//     PlcTask Inputs/G_IO.arDI[68]/Ch[15] <-> Module 4 (GL20-1600END)/1600END input-bit maping/Digital input CH2-bit7
//     PlcTask Inputs/G_IO.arDI[68]/Ch[1] <-> Module 4 (GL20-1600END)/1600END input-bit maping/Digital input CH1-bit1
//     PlcTask Inputs/G_IO.arDI[68]/Ch[2] <-> Module 4 (GL20-1600END)/1600END input-bit maping/Digital input CH1-bit2
//     PlcTask Inputs/G_IO.arDI[68]/Ch[3] <-> Module 4 (GL20-1600END)/1600END input-bit maping/Digital input CH1-bit3
//     PlcTask Inputs/G_IO.arDI[68]/Ch[4] <-> Module 4 (GL20-1600END)/1600END input-bit maping/Digital input CH1-bit4
//     PlcTask Inputs/G_IO.arDI[68]/Ch[5] <-> Module 4 (GL20-1600END)/1600END input-bit maping/Digital input CH1-bit5
//     PlcTask Inputs/G_IO.arDI[68]/Ch[6] <-> Module 4 (GL20-1600END)/1600END input-bit maping/Digital input CH1-bit6
//     PlcTask Inputs/G_IO.arDI[68]/Ch[7] <-> Module 4 (GL20-1600END)/1600END input-bit maping/Digital input CH1-bit7
//     PlcTask Inputs/G_IO.arDI[68]/Ch[8] <-> Module 4 (GL20-1600END)/1600END input-bit maping/Digital input CH2-bit0
//     PlcTask Inputs/G_IO.arDI[68]/Ch[9] <-> Module 4 (GL20-1600END)/1600END input-bit maping/Digital input CH2-bit1
//     PlcTask Inputs/G_IO.arDI[69]/Ch[0] <-> Module 5 (GL20-1600END)/1600END input-bit maping/Digital input CH1-bit0
//     PlcTask Inputs/G_IO.arDI[69]/Ch[10] <-> Module 5 (GL20-1600END)/1600END input-bit maping/Digital input CH2-bit2
//     PlcTask Inputs/G_IO.arDI[69]/Ch[11] <-> Module 5 (GL20-1600END)/1600END input-bit maping/Digital input CH2-bit3
//     PlcTask Inputs/G_IO.arDI[69]/Ch[12] <-> Module 5 (GL20-1600END)/1600END input-bit maping/Digital input CH2-bit4
//     PlcTask Inputs/G_IO.arDI[69]/Ch[13] <-> Module 5 (GL20-1600END)/1600END input-bit maping/Digital input CH2-bit5
//     PlcTask Inputs/G_IO.arDI[69]/Ch[14] <-> Module 5 (GL20-1600END)/1600END input-bit maping/Digital input CH2-bit6
//     PlcTask Inputs/G_IO.arDI[69]/Ch[15] <-> Module 5 (GL20-1600END)/1600END input-bit maping/Digital input CH2-bit7
//     PlcTask Inputs/G_IO.arDI[69]/Ch[1] <-> Module 5 (GL20-1600END)/1600END input-bit maping/Digital input CH1-bit1
//     PlcTask Inputs/G_IO.arDI[69]/Ch[2] <-> Module 5 (GL20-1600END)/1600END input-bit maping/Digital input CH1-bit2
//     PlcTask Inputs/G_IO.arDI[69]/Ch[3] <-> Module 5 (GL20-1600END)/1600END input-bit maping/Digital input CH1-bit3
//     PlcTask Inputs/G_IO.arDI[69]/Ch[4] <-> Module 5 (GL20-1600END)/1600END input-bit maping/Digital input CH1-bit4
//     PlcTask Inputs/G_IO.arDI[69]/Ch[5] <-> Module 5 (GL20-1600END)/1600END input-bit maping/Digital input CH1-bit5
//     PlcTask Inputs/G_IO.arDI[69]/Ch[6] <-> Module 5 (GL20-1600END)/1600END input-bit maping/Digital input CH1-bit6
//     PlcTask Inputs/G_IO.arDI[69]/Ch[7] <-> Module 5 (GL20-1600END)/1600END input-bit maping/Digital input CH1-bit7
//     PlcTask Inputs/G_IO.arDI[69]/Ch[8] <-> Module 5 (GL20-1600END)/1600END input-bit maping/Digital input CH2-bit0
//     PlcTask Inputs/G_IO.arDI[69]/Ch[9] <-> Module 5 (GL20-1600END)/1600END input-bit maping/Digital input CH2-bit1
//     PlcTask Outputs/G_IO.arDO[62]/Ch[0] <-> Module 6 (GL20-0016ETP)/0016ETP Output-bit maping/Digital output CH1-bit0
//     PlcTask Outputs/G_IO.arDO[62]/Ch[10] <-> Module 6 (GL20-0016ETP)/0016ETP Output-bit maping/Digital output CH2-bit2
//     PlcTask Outputs/G_IO.arDO[62]/Ch[11] <-> Module 6 (GL20-0016ETP)/0016ETP Output-bit maping/Digital output CH2-bit3
//     PlcTask Outputs/G_IO.arDO[62]/Ch[12] <-> Module 6 (GL20-0016ETP)/0016ETP Output-bit maping/Digital output CH2-bit4
//     PlcTask Outputs/G_IO.arDO[62]/Ch[13] <-> Module 6 (GL20-0016ETP)/0016ETP Output-bit maping/Digital output CH2-bit5
//     PlcTask Outputs/G_IO.arDO[62]/Ch[14] <-> Module 6 (GL20-0016ETP)/0016ETP Output-bit maping/Digital output CH2-bit6
//     PlcTask Outputs/G_IO.arDO[62]/Ch[15] <-> Module 6 (GL20-0016ETP)/0016ETP Output-bit maping/Digital output CH2-bit7
//     PlcTask Outputs/G_IO.arDO[62]/Ch[1] <-> Module 6 (GL20-0016ETP)/0016ETP Output-bit maping/Digital output CH1-bit1
//     PlcTask Outputs/G_IO.arDO[62]/Ch[2] <-> Module 6 (GL20-0016ETP)/0016ETP Output-bit maping/Digital output CH1-bit2
//     PlcTask Outputs/G_IO.arDO[62]/Ch[3] <-> Module 6 (GL20-0016ETP)/0016ETP Output-bit maping/Digital output CH1-bit3
//     PlcTask Outputs/G_IO.arDO[62]/Ch[4] <-> Module 6 (GL20-0016ETP)/0016ETP Output-bit maping/Digital output CH1-bit4
//     PlcTask Outputs/G_IO.arDO[62]/Ch[5] <-> Module 6 (GL20-0016ETP)/0016ETP Output-bit maping/Digital output CH1-bit5
//     PlcTask Outputs/G_IO.arDO[62]/Ch[6] <-> Module 6 (GL20-0016ETP)/0016ETP Output-bit maping/Digital output CH1-bit6
//     PlcTask Outputs/G_IO.arDO[62]/Ch[7] <-> Module 6 (GL20-0016ETP)/0016ETP Output-bit maping/Digital output CH1-bit7
//     PlcTask Outputs/G_IO.arDO[62]/Ch[8] <-> Module 6 (GL20-0016ETP)/0016ETP Output-bit maping/Digital output CH2-bit0
//     PlcTask Outputs/G_IO.arDO[62]/Ch[9] <-> Module 6 (GL20-0016ETP)/0016ETP Output-bit maping/Digital output CH2-bit1
//     PlcTask Outputs/G_IO.arDO[63]/Ch[0] <-> Module 7 (GL20-0016ETP)/0016ETP Output-bit maping/Digital output CH1-bit0
//     PlcTask Outputs/G_IO.arDO[63]/Ch[10] <-> Module 7 (GL20-0016ETP)/0016ETP Output-bit maping/Digital output CH2-bit2
//     PlcTask Outputs/G_IO.arDO[63]/Ch[11] <-> Module 7 (GL20-0016ETP)/0016ETP Output-bit maping/Digital output CH2-bit3
//     PlcTask Outputs/G_IO.arDO[63]/Ch[12] <-> Module 7 (GL20-0016ETP)/0016ETP Output-bit maping/Digital output CH2-bit4
//     PlcTask Outputs/G_IO.arDO[63]/Ch[13] <-> Module 7 (GL20-0016ETP)/0016ETP Output-bit maping/Digital output CH2-bit5
//     PlcTask Outputs/G_IO.arDO[63]/Ch[14] <-> Module 7 (GL20-0016ETP)/0016ETP Output-bit maping/Digital output CH2-bit6
//     PlcTask Outputs/G_IO.arDO[63]/Ch[15] <-> Module 7 (GL20-0016ETP)/0016ETP Output-bit maping/Digital output CH2-bit7
//     PlcTask Outputs/G_IO.arDO[63]/Ch[1] <-> Module 7 (GL20-0016ETP)/0016ETP Output-bit maping/Digital output CH1-bit1
//     PlcTask Outputs/G_IO.arDO[63]/Ch[2] <-> Module 7 (GL20-0016ETP)/0016ETP Output-bit maping/Digital output CH1-bit2
//     PlcTask Outputs/G_IO.arDO[63]/Ch[3] <-> Module 7 (GL20-0016ETP)/0016ETP Output-bit maping/Digital output CH1-bit3
//     PlcTask Outputs/G_IO.arDO[63]/Ch[4] <-> Module 7 (GL20-0016ETP)/0016ETP Output-bit maping/Digital output CH1-bit4
//     PlcTask Outputs/G_IO.arDO[63]/Ch[5] <-> Module 7 (GL20-0016ETP)/0016ETP Output-bit maping/Digital output CH1-bit5
//     PlcTask Outputs/G_IO.arDO[63]/Ch[6] <-> Module 7 (GL20-0016ETP)/0016ETP Output-bit maping/Digital output CH1-bit6
//     PlcTask Outputs/G_IO.arDO[63]/Ch[7] <-> Module 7 (GL20-0016ETP)/0016ETP Output-bit maping/Digital output CH1-bit7
//     PlcTask Outputs/G_IO.arDO[63]/Ch[8] <-> Module 7 (GL20-0016ETP)/0016ETP Output-bit maping/Digital output CH2-bit0
//     PlcTask Outputs/G_IO.arDO[63]/Ch[9] <-> Module 7 (GL20-0016ETP)/0016ETP Output-bit maping/Digital output CH2-bit1
//   kittingDeca/kittingDeca Instance <-> pm side/pm6_7_innerConv
//     PlcTask Inputs/GVL.pm[6].inConv.belt[0].fbconverter.running_freq <-> Axis#1 Iutputs/Axis1 Running frequency
//     PlcTask Inputs/GVL.pm[6].inConv.belt[1].fbconverter.running_freq <-> Axis#2 Iutputs/Axis2 Running frequency
//     PlcTask Inputs/GVL.pm[6].inConv.belt[2].fbconverter.running_freq <-> Axis#3 Iutputs/Axis3 Running frequency
//     PlcTask Inputs/GVL.pm[7].inConv.belt[0].fbconverter.running_freq <-> Axis#4 Iutputs/Axis4 Running frequency
//     PlcTask Inputs/GVL.pm[7].inConv.belt[1].fbconverter.running_freq <-> Axis#5 Iutputs/Axis5 Running frequency
//     PlcTask Inputs/GVL.pm[7].inConv.belt[2].fbconverter.running_freq <-> Axis#6 Iutputs/Axis6 Running frequency
//     PlcTask Inputs/GVL.pm[6].inConv.belt[0].fbconverter.status <-> Axis#1 Iutputs/Axis1 AC drive running status word 2
//     PlcTask Inputs/GVL.pm[6].inConv.belt[1].fbconverter.status <-> Axis#2 Iutputs/Axis2 AC drive running status word 2
//     PlcTask Inputs/GVL.pm[6].inConv.belt[2].fbconverter.status <-> Axis#3 Iutputs/Axis3 AC drive running status word 2
//     PlcTask Inputs/GVL.pm[7].inConv.belt[0].fbconverter.status <-> Axis#4 Iutputs/Axis4 AC drive running status word 2
//     PlcTask Inputs/GVL.pm[7].inConv.belt[1].fbconverter.status <-> Axis#5 Iutputs/Axis5 AC drive running status word 2
//     PlcTask Inputs/GVL.pm[7].inConv.belt[2].fbconverter.status <-> Axis#6 Iutputs/Axis6 AC drive running status word 2
//     PlcTask Outputs/GVL.pm[6].inConv.belt[0].fbconverter.cmd <-> Axis#1 Outputs/Axis1 Communication control command
//     PlcTask Outputs/GVL.pm[6].inConv.belt[1].fbconverter.cmd <-> Axis#2 Outputs/Axis2 Communication control command
//     PlcTask Outputs/GVL.pm[6].inConv.belt[2].fbconverter.cmd <-> Axis#3 Outputs/Axis3 Communication control command
//     PlcTask Outputs/GVL.pm[7].inConv.belt[0].fbconverter.cmd <-> Axis#4 Outputs/Axis4 Communication control command
//     PlcTask Outputs/GVL.pm[7].inConv.belt[1].fbconverter.cmd <-> Axis#5 Outputs/Axis5 Communication control command
//     PlcTask Outputs/GVL.pm[7].inConv.belt[2].fbconverter.cmd <-> Axis#6 Outputs/Axis6 Communication control command
//     PlcTask Outputs/GVL.pm[6].inConv.belt[0].fbconverter.freq <-> Axis#1 Outputs/Axis1 Frequency set through communication
//     PlcTask Outputs/GVL.pm[6].inConv.belt[1].fbconverter.freq <-> Axis#2 Outputs/Axis2 Frequency set through communication
//     PlcTask Outputs/GVL.pm[6].inConv.belt[2].fbconverter.freq <-> Axis#3 Outputs/Axis3 Frequency set through communication
//     PlcTask Outputs/GVL.pm[7].inConv.belt[0].fbconverter.freq <-> Axis#4 Outputs/Axis4 Frequency set through communication
//     PlcTask Outputs/GVL.pm[7].inConv.belt[1].fbconverter.freq <-> Axis#5 Outputs/Axis5 Frequency set through communication
//     PlcTask Outputs/GVL.pm[7].inConv.belt[2].fbconverter.freq <-> Axis#6 Outputs/Axis6 Frequency set through communication
//   kittingDeca/kittingDeca Instance <-> pm side/pm6_7_outerConv
//     PlcTask Inputs/GVL.pm[6].outConv.belt[0].fbconverter.running_freq <-> Axis#1 Iutputs/Axis1 Running frequency
//     PlcTask Inputs/GVL.pm[6].outConv.belt[1].fbconverter.running_freq <-> Axis#2 Iutputs/Axis2 Running frequency
//     PlcTask Inputs/GVL.pm[7].outConv.belt[0].fbconverter.running_freq <-> Axis#3 Iutputs/Axis3 Running frequency
//     PlcTask Inputs/GVL.pm[7].outConv.belt[1].fbconverter.running_freq <-> Axis#4 Iutputs/Axis4 Running frequency
//     PlcTask Inputs/GVL.pm[6].outConv.belt[0].fbconverter.status <-> Axis#1 Iutputs/Axis1 AC drive running status word 2
//     PlcTask Inputs/GVL.pm[6].outConv.belt[1].fbconverter.status <-> Axis#2 Iutputs/Axis2 AC drive running status word 2
//     PlcTask Inputs/GVL.pm[7].outConv.belt[0].fbconverter.status <-> Axis#3 Iutputs/Axis3 AC drive running status word 2
//     PlcTask Inputs/GVL.pm[7].outConv.belt[1].fbconverter.status <-> Axis#4 Iutputs/Axis4 AC drive running status word 2
//     PlcTask Outputs/GVL.pm[6].outConv.belt[0].fbconverter.cmd <-> Axis#1 Outputs/Axis1 Communication control command
//     PlcTask Outputs/GVL.pm[6].outConv.belt[1].fbconverter.cmd <-> Axis#2 Outputs/Axis2 Communication control command
//     PlcTask Outputs/GVL.pm[7].outConv.belt[0].fbconverter.cmd <-> Axis#3 Outputs/Axis3 Communication control command
//     PlcTask Outputs/GVL.pm[7].outConv.belt[1].fbconverter.cmd <-> Axis#4 Outputs/Axis4 Communication control command
//     PlcTask Outputs/GVL.pm[6].outConv.belt[0].fbconverter.freq <-> Axis#1 Outputs/Axis1 Frequency set through communication
//     PlcTask Outputs/GVL.pm[6].outConv.belt[1].fbconverter.freq <-> Axis#2 Outputs/Axis2 Frequency set through communication
//     PlcTask Outputs/GVL.pm[7].outConv.belt[0].fbconverter.freq <-> Axis#3 Outputs/Axis3 Frequency set through communication
//     PlcTask Outputs/GVL.pm[7].outConv.belt[1].fbconverter.freq <-> Axis#4 Outputs/Axis4 Frequency set through communication
//   kittingDeca/kittingDeca Instance <-> pm side/pm8_9_dio
//     PlcTask Inputs/G_IO.arDI[70]/Ch[0] <-> Module 1 (GL20-1600END)/1600END input-bit maping/Digital input CH1-bit0
//     PlcTask Inputs/G_IO.arDI[70]/Ch[10] <-> Module 1 (GL20-1600END)/1600END input-bit maping/Digital input CH2-bit2
//     PlcTask Inputs/G_IO.arDI[70]/Ch[11] <-> Module 1 (GL20-1600END)/1600END input-bit maping/Digital input CH2-bit3
//     PlcTask Inputs/G_IO.arDI[70]/Ch[12] <-> Module 1 (GL20-1600END)/1600END input-bit maping/Digital input CH2-bit4
//     PlcTask Inputs/G_IO.arDI[70]/Ch[13] <-> Module 1 (GL20-1600END)/1600END input-bit maping/Digital input CH2-bit5
//     PlcTask Inputs/G_IO.arDI[70]/Ch[14] <-> Module 1 (GL20-1600END)/1600END input-bit maping/Digital input CH2-bit6
//     PlcTask Inputs/G_IO.arDI[70]/Ch[15] <-> Module 1 (GL20-1600END)/1600END input-bit maping/Digital input CH2-bit7
//     PlcTask Inputs/G_IO.arDI[70]/Ch[1] <-> Module 1 (GL20-1600END)/1600END input-bit maping/Digital input CH1-bit1
//     PlcTask Inputs/G_IO.arDI[70]/Ch[2] <-> Module 1 (GL20-1600END)/1600END input-bit maping/Digital input CH1-bit2
//     PlcTask Inputs/G_IO.arDI[70]/Ch[3] <-> Module 1 (GL20-1600END)/1600END input-bit maping/Digital input CH1-bit3
//     PlcTask Inputs/G_IO.arDI[70]/Ch[4] <-> Module 1 (GL20-1600END)/1600END input-bit maping/Digital input CH1-bit4
//     PlcTask Inputs/G_IO.arDI[70]/Ch[5] <-> Module 1 (GL20-1600END)/1600END input-bit maping/Digital input CH1-bit5
//     PlcTask Inputs/G_IO.arDI[70]/Ch[6] <-> Module 1 (GL20-1600END)/1600END input-bit maping/Digital input CH1-bit6
//     PlcTask Inputs/G_IO.arDI[70]/Ch[7] <-> Module 1 (GL20-1600END)/1600END input-bit maping/Digital input CH1-bit7
//     PlcTask Inputs/G_IO.arDI[70]/Ch[8] <-> Module 1 (GL20-1600END)/1600END input-bit maping/Digital input CH2-bit0
//     PlcTask Inputs/G_IO.arDI[70]/Ch[9] <-> Module 1 (GL20-1600END)/1600END input-bit maping/Digital input CH2-bit1
//     PlcTask Inputs/G_IO.arDI[71]/Ch[0] <-> Module 2 (GL20-1600END)/1600END input-bit maping/Digital input CH1-bit0
//     PlcTask Inputs/G_IO.arDI[71]/Ch[10] <-> Module 2 (GL20-1600END)/1600END input-bit maping/Digital input CH2-bit2
//     PlcTask Inputs/G_IO.arDI[71]/Ch[11] <-> Module 2 (GL20-1600END)/1600END input-bit maping/Digital input CH2-bit3
//     PlcTask Inputs/G_IO.arDI[71]/Ch[12] <-> Module 2 (GL20-1600END)/1600END input-bit maping/Digital input CH2-bit4
//     PlcTask Inputs/G_IO.arDI[71]/Ch[13] <-> Module 2 (GL20-1600END)/1600END input-bit maping/Digital input CH2-bit5
//     PlcTask Inputs/G_IO.arDI[71]/Ch[14] <-> Module 2 (GL20-1600END)/1600END input-bit maping/Digital input CH2-bit6
//     PlcTask Inputs/G_IO.arDI[71]/Ch[15] <-> Module 2 (GL20-1600END)/1600END input-bit maping/Digital input CH2-bit7
//     PlcTask Inputs/G_IO.arDI[71]/Ch[1] <-> Module 2 (GL20-1600END)/1600END input-bit maping/Digital input CH1-bit1
//     PlcTask Inputs/G_IO.arDI[71]/Ch[2] <-> Module 2 (GL20-1600END)/1600END input-bit maping/Digital input CH1-bit2
//     PlcTask Inputs/G_IO.arDI[71]/Ch[3] <-> Module 2 (GL20-1600END)/1600END input-bit maping/Digital input CH1-bit3
//     PlcTask Inputs/G_IO.arDI[71]/Ch[4] <-> Module 2 (GL20-1600END)/1600END input-bit maping/Digital input CH1-bit4
//     PlcTask Inputs/G_IO.arDI[71]/Ch[5] <-> Module 2 (GL20-1600END)/1600END input-bit maping/Digital input CH1-bit5
//     PlcTask Inputs/G_IO.arDI[71]/Ch[6] <-> Module 2 (GL20-1600END)/1600END input-bit maping/Digital input CH1-bit6
//     PlcTask Inputs/G_IO.arDI[71]/Ch[7] <-> Module 2 (GL20-1600END)/1600END input-bit maping/Digital input CH1-bit7
//     PlcTask Inputs/G_IO.arDI[71]/Ch[8] <-> Module 2 (GL20-1600END)/1600END input-bit maping/Digital input CH2-bit0
//     PlcTask Inputs/G_IO.arDI[71]/Ch[9] <-> Module 2 (GL20-1600END)/1600END input-bit maping/Digital input CH2-bit1
//     PlcTask Inputs/G_IO.arDI[72]/Ch[0] <-> Module 3 (GL20-1600END)/1600END input-bit maping/Digital input CH1-bit0
//     PlcTask Inputs/G_IO.arDI[72]/Ch[10] <-> Module 3 (GL20-1600END)/1600END input-bit maping/Digital input CH2-bit2
//     PlcTask Inputs/G_IO.arDI[72]/Ch[11] <-> Module 3 (GL20-1600END)/1600END input-bit maping/Digital input CH2-bit3
//     PlcTask Inputs/G_IO.arDI[72]/Ch[12] <-> Module 3 (GL20-1600END)/1600END input-bit maping/Digital input CH2-bit4
//     PlcTask Inputs/G_IO.arDI[72]/Ch[13] <-> Module 3 (GL20-1600END)/1600END input-bit maping/Digital input CH2-bit5
//     PlcTask Inputs/G_IO.arDI[72]/Ch[14] <-> Module 3 (GL20-1600END)/1600END input-bit maping/Digital input CH2-bit6
//     PlcTask Inputs/G_IO.arDI[72]/Ch[15] <-> Module 3 (GL20-1600END)/1600END input-bit maping/Digital input CH2-bit7
//     PlcTask Inputs/G_IO.arDI[72]/Ch[1] <-> Module 3 (GL20-1600END)/1600END input-bit maping/Digital input CH1-bit1
//     PlcTask Inputs/G_IO.arDI[72]/Ch[2] <-> Module 3 (GL20-1600END)/1600END input-bit maping/Digital input CH1-bit2
//     PlcTask Inputs/G_IO.arDI[72]/Ch[3] <-> Module 3 (GL20-1600END)/1600END input-bit maping/Digital input CH1-bit3
//     PlcTask Inputs/G_IO.arDI[72]/Ch[4] <-> Module 3 (GL20-1600END)/1600END input-bit maping/Digital input CH1-bit4
//     PlcTask Inputs/G_IO.arDI[72]/Ch[5] <-> Module 3 (GL20-1600END)/1600END input-bit maping/Digital input CH1-bit5
//     PlcTask Inputs/G_IO.arDI[72]/Ch[6] <-> Module 3 (GL20-1600END)/1600END input-bit maping/Digital input CH1-bit6
//     PlcTask Inputs/G_IO.arDI[72]/Ch[7] <-> Module 3 (GL20-1600END)/1600END input-bit maping/Digital input CH1-bit7
//     PlcTask Inputs/G_IO.arDI[72]/Ch[8] <-> Module 3 (GL20-1600END)/1600END input-bit maping/Digital input CH2-bit0
//     PlcTask Inputs/G_IO.arDI[72]/Ch[9] <-> Module 3 (GL20-1600END)/1600END input-bit maping/Digital input CH2-bit1
//     PlcTask Inputs/G_IO.arDI[73]/Ch[0] <-> Module 4 (GL20-1600END)/1600END input-bit maping/Digital input CH1-bit0
//     PlcTask Inputs/G_IO.arDI[73]/Ch[10] <-> Module 4 (GL20-1600END)/1600END input-bit maping/Digital input CH2-bit2
//     PlcTask Inputs/G_IO.arDI[73]/Ch[11] <-> Module 4 (GL20-1600END)/1600END input-bit maping/Digital input CH2-bit3
//     PlcTask Inputs/G_IO.arDI[73]/Ch[12] <-> Module 4 (GL20-1600END)/1600END input-bit maping/Digital input CH2-bit4
//     PlcTask Inputs/G_IO.arDI[73]/Ch[13] <-> Module 4 (GL20-1600END)/1600END input-bit maping/Digital input CH2-bit5
//     PlcTask Inputs/G_IO.arDI[73]/Ch[14] <-> Module 4 (GL20-1600END)/1600END input-bit maping/Digital input CH2-bit6
//     PlcTask Inputs/G_IO.arDI[73]/Ch[15] <-> Module 4 (GL20-1600END)/1600END input-bit maping/Digital input CH2-bit7
//     PlcTask Inputs/G_IO.arDI[73]/Ch[1] <-> Module 4 (GL20-1600END)/1600END input-bit maping/Digital input CH1-bit1
//     PlcTask Inputs/G_IO.arDI[73]/Ch[2] <-> Module 4 (GL20-1600END)/1600END input-bit maping/Digital input CH1-bit2
//     PlcTask Inputs/G_IO.arDI[73]/Ch[3] <-> Module 4 (GL20-1600END)/1600END input-bit maping/Digital input CH1-bit3
//     PlcTask Inputs/G_IO.arDI[73]/Ch[4] <-> Module 4 (GL20-1600END)/1600END input-bit maping/Digital input CH1-bit4
//     PlcTask Inputs/G_IO.arDI[73]/Ch[5] <-> Module 4 (GL20-1600END)/1600END input-bit maping/Digital input CH1-bit5
//     PlcTask Inputs/G_IO.arDI[73]/Ch[6] <-> Module 4 (GL20-1600END)/1600END input-bit maping/Digital input CH1-bit6
//     PlcTask Inputs/G_IO.arDI[73]/Ch[7] <-> Module 4 (GL20-1600END)/1600END input-bit maping/Digital input CH1-bit7
//     PlcTask Inputs/G_IO.arDI[73]/Ch[8] <-> Module 4 (GL20-1600END)/1600END input-bit maping/Digital input CH2-bit0
//     PlcTask Inputs/G_IO.arDI[73]/Ch[9] <-> Module 4 (GL20-1600END)/1600END input-bit maping/Digital input CH2-bit1
//     PlcTask Inputs/G_IO.arDI[74]/Ch[0] <-> Module 5 (GL20-1600END)/1600END input-bit maping/Digital input CH1-bit0
//     PlcTask Inputs/G_IO.arDI[74]/Ch[10] <-> Module 5 (GL20-1600END)/1600END input-bit maping/Digital input CH2-bit2
//     PlcTask Inputs/G_IO.arDI[74]/Ch[11] <-> Module 5 (GL20-1600END)/1600END input-bit maping/Digital input CH2-bit3
//     PlcTask Inputs/G_IO.arDI[74]/Ch[12] <-> Module 5 (GL20-1600END)/1600END input-bit maping/Digital input CH2-bit4
//     PlcTask Inputs/G_IO.arDI[74]/Ch[13] <-> Module 5 (GL20-1600END)/1600END input-bit maping/Digital input CH2-bit5
//     PlcTask Inputs/G_IO.arDI[74]/Ch[14] <-> Module 5 (GL20-1600END)/1600END input-bit maping/Digital input CH2-bit6
//     PlcTask Inputs/G_IO.arDI[74]/Ch[15] <-> Module 5 (GL20-1600END)/1600END input-bit maping/Digital input CH2-bit7
//     PlcTask Inputs/G_IO.arDI[74]/Ch[1] <-> Module 5 (GL20-1600END)/1600END input-bit maping/Digital input CH1-bit1
//     PlcTask Inputs/G_IO.arDI[74]/Ch[2] <-> Module 5 (GL20-1600END)/1600END input-bit maping/Digital input CH1-bit2
//     PlcTask Inputs/G_IO.arDI[74]/Ch[3] <-> Module 5 (GL20-1600END)/1600END input-bit maping/Digital input CH1-bit3
//     PlcTask Inputs/G_IO.arDI[74]/Ch[4] <-> Module 5 (GL20-1600END)/1600END input-bit maping/Digital input CH1-bit4
//     PlcTask Inputs/G_IO.arDI[74]/Ch[5] <-> Module 5 (GL20-1600END)/1600END input-bit maping/Digital input CH1-bit5
//     PlcTask Inputs/G_IO.arDI[74]/Ch[6] <-> Module 5 (GL20-1600END)/1600END input-bit maping/Digital input CH1-bit6
//     PlcTask Inputs/G_IO.arDI[74]/Ch[7] <-> Module 5 (GL20-1600END)/1600END input-bit maping/Digital input CH1-bit7
//     PlcTask Inputs/G_IO.arDI[74]/Ch[8] <-> Module 5 (GL20-1600END)/1600END input-bit maping/Digital input CH2-bit0
//     PlcTask Inputs/G_IO.arDI[74]/Ch[9] <-> Module 5 (GL20-1600END)/1600END input-bit maping/Digital input CH2-bit1
//     PlcTask Outputs/G_IO.arDO[66]/Ch[0] <-> Module 6 (GL20-0016ETP)/0016ETP Output-bit maping/Digital output CH1-bit0
//     PlcTask Outputs/G_IO.arDO[66]/Ch[10] <-> Module 6 (GL20-0016ETP)/0016ETP Output-bit maping/Digital output CH2-bit2
//     PlcTask Outputs/G_IO.arDO[66]/Ch[11] <-> Module 6 (GL20-0016ETP)/0016ETP Output-bit maping/Digital output CH2-bit3
//     PlcTask Outputs/G_IO.arDO[66]/Ch[12] <-> Module 6 (GL20-0016ETP)/0016ETP Output-bit maping/Digital output CH2-bit4
//     PlcTask Outputs/G_IO.arDO[66]/Ch[13] <-> Module 6 (GL20-0016ETP)/0016ETP Output-bit maping/Digital output CH2-bit5
//     PlcTask Outputs/G_IO.arDO[66]/Ch[14] <-> Module 6 (GL20-0016ETP)/0016ETP Output-bit maping/Digital output CH2-bit6
//     PlcTask Outputs/G_IO.arDO[66]/Ch[15] <-> Module 6 (GL20-0016ETP)/0016ETP Output-bit maping/Digital output CH2-bit7
//     PlcTask Outputs/G_IO.arDO[66]/Ch[1] <-> Module 6 (GL20-0016ETP)/0016ETP Output-bit maping/Digital output CH1-bit1
//     PlcTask Outputs/G_IO.arDO[66]/Ch[2] <-> Module 6 (GL20-0016ETP)/0016ETP Output-bit maping/Digital output CH1-bit2
//     PlcTask Outputs/G_IO.arDO[66]/Ch[3] <-> Module 6 (GL20-0016ETP)/0016ETP Output-bit maping/Digital output CH1-bit3
//     PlcTask Outputs/G_IO.arDO[66]/Ch[4] <-> Module 6 (GL20-0016ETP)/0016ETP Output-bit maping/Digital output CH1-bit4
//     PlcTask Outputs/G_IO.arDO[66]/Ch[5] <-> Module 6 (GL20-0016ETP)/0016ETP Output-bit maping/Digital output CH1-bit5
//     PlcTask Outputs/G_IO.arDO[66]/Ch[6] <-> Module 6 (GL20-0016ETP)/0016ETP Output-bit maping/Digital output CH1-bit6
//     PlcTask Outputs/G_IO.arDO[66]/Ch[7] <-> Module 6 (GL20-0016ETP)/0016ETP Output-bit maping/Digital output CH1-bit7
//     PlcTask Outputs/G_IO.arDO[66]/Ch[8] <-> Module 6 (GL20-0016ETP)/0016ETP Output-bit maping/Digital output CH2-bit0
//     PlcTask Outputs/G_IO.arDO[66]/Ch[9] <-> Module 6 (GL20-0016ETP)/0016ETP Output-bit maping/Digital output CH2-bit1
//     PlcTask Outputs/G_IO.arDO[67]/Ch[0] <-> Module 7 (GL20-0016ETP)/0016ETP Output-bit maping/Digital output CH1-bit0
//     PlcTask Outputs/G_IO.arDO[67]/Ch[10] <-> Module 7 (GL20-0016ETP)/0016ETP Output-bit maping/Digital output CH2-bit2
//     PlcTask Outputs/G_IO.arDO[67]/Ch[11] <-> Module 7 (GL20-0016ETP)/0016ETP Output-bit maping/Digital output CH2-bit3
//     PlcTask Outputs/G_IO.arDO[67]/Ch[12] <-> Module 7 (GL20-0016ETP)/0016ETP Output-bit maping/Digital output CH2-bit4
//     PlcTask Outputs/G_IO.arDO[67]/Ch[13] <-> Module 7 (GL20-0016ETP)/0016ETP Output-bit maping/Digital output CH2-bit5
//     PlcTask Outputs/G_IO.arDO[67]/Ch[14] <-> Module 7 (GL20-0016ETP)/0016ETP Output-bit maping/Digital output CH2-bit6
//     PlcTask Outputs/G_IO.arDO[67]/Ch[15] <-> Module 7 (GL20-0016ETP)/0016ETP Output-bit maping/Digital output CH2-bit7
//     PlcTask Outputs/G_IO.arDO[67]/Ch[1] <-> Module 7 (GL20-0016ETP)/0016ETP Output-bit maping/Digital output CH1-bit1
//     PlcTask Outputs/G_IO.arDO[67]/Ch[2] <-> Module 7 (GL20-0016ETP)/0016ETP Output-bit maping/Digital output CH1-bit2
//     PlcTask Outputs/G_IO.arDO[67]/Ch[3] <-> Module 7 (GL20-0016ETP)/0016ETP Output-bit maping/Digital output CH1-bit3
//     PlcTask Outputs/G_IO.arDO[67]/Ch[4] <-> Module 7 (GL20-0016ETP)/0016ETP Output-bit maping/Digital output CH1-bit4
//     PlcTask Outputs/G_IO.arDO[67]/Ch[5] <-> Module 7 (GL20-0016ETP)/0016ETP Output-bit maping/Digital output CH1-bit5
//     PlcTask Outputs/G_IO.arDO[67]/Ch[6] <-> Module 7 (GL20-0016ETP)/0016ETP Output-bit maping/Digital output CH1-bit6
//     PlcTask Outputs/G_IO.arDO[67]/Ch[7] <-> Module 7 (GL20-0016ETP)/0016ETP Output-bit maping/Digital output CH1-bit7
//     PlcTask Outputs/G_IO.arDO[67]/Ch[8] <-> Module 7 (GL20-0016ETP)/0016ETP Output-bit maping/Digital output CH2-bit0
//     PlcTask Outputs/G_IO.arDO[67]/Ch[9] <-> Module 7 (GL20-0016ETP)/0016ETP Output-bit maping/Digital output CH2-bit1
//   kittingDeca/kittingDeca Instance <-> pm side/pm8_9_innerConv
//     PlcTask Inputs/GVL.pm[8].inConv.belt[0].fbconverter.running_freq <-> Axis#1 Iutputs/Axis1 Running frequency
//     PlcTask Inputs/GVL.pm[8].inConv.belt[1].fbconverter.running_freq <-> Axis#2 Iutputs/Axis2 Running frequency
//     PlcTask Inputs/GVL.pm[8].inConv.belt[2].fbconverter.running_freq <-> Axis#3 Iutputs/Axis3 Running frequency
//     PlcTask Inputs/GVL.pm[9].inConv.belt[0].fbconverter.running_freq <-> Axis#4 Iutputs/Axis4 Running frequency
//     PlcTask Inputs/GVL.pm[9].inConv.belt[1].fbconverter.running_freq <-> Axis#5 Iutputs/Axis5 Running frequency
//     PlcTask Inputs/GVL.pm[9].inConv.belt[2].fbconverter.running_freq <-> Axis#6 Iutputs/Axis6 Running frequency
//     PlcTask Inputs/GVL.pm[8].inConv.belt[0].fbconverter.status <-> Axis#1 Iutputs/Axis1 AC drive running status word 2
//     PlcTask Inputs/GVL.pm[8].inConv.belt[1].fbconverter.status <-> Axis#2 Iutputs/Axis2 AC drive running status word 2
//     PlcTask Inputs/GVL.pm[8].inConv.belt[2].fbconverter.status <-> Axis#3 Iutputs/Axis3 AC drive running status word 2
//     PlcTask Inputs/GVL.pm[9].inConv.belt[0].fbconverter.status <-> Axis#4 Iutputs/Axis4 AC drive running status word 2
//     PlcTask Inputs/GVL.pm[9].inConv.belt[1].fbconverter.status <-> Axis#5 Iutputs/Axis5 AC drive running status word 2
//     PlcTask Inputs/GVL.pm[9].inConv.belt[2].fbconverter.status <-> Axis#6 Iutputs/Axis6 AC drive running status word 2
//     PlcTask Outputs/GVL.pm[8].inConv.belt[0].fbconverter.cmd <-> Axis#1 Outputs/Axis1 Communication control command
//     PlcTask Outputs/GVL.pm[8].inConv.belt[1].fbconverter.cmd <-> Axis#2 Outputs/Axis2 Communication control command
//     PlcTask Outputs/GVL.pm[8].inConv.belt[2].fbconverter.cmd <-> Axis#3 Outputs/Axis3 Communication control command
//     PlcTask Outputs/GVL.pm[9].inConv.belt[0].fbconverter.cmd <-> Axis#4 Outputs/Axis4 Communication control command
//     PlcTask Outputs/GVL.pm[9].inConv.belt[1].fbconverter.cmd <-> Axis#5 Outputs/Axis5 Communication control command
//     PlcTask Outputs/GVL.pm[9].inConv.belt[2].fbconverter.cmd <-> Axis#6 Outputs/Axis6 Communication control command
//     PlcTask Outputs/GVL.pm[8].inConv.belt[0].fbconverter.freq <-> Axis#1 Outputs/Axis1 Frequency set through communication
//     PlcTask Outputs/GVL.pm[8].inConv.belt[1].fbconverter.freq <-> Axis#2 Outputs/Axis2 Frequency set through communication
//     PlcTask Outputs/GVL.pm[8].inConv.belt[2].fbconverter.freq <-> Axis#3 Outputs/Axis3 Frequency set through communication
//     PlcTask Outputs/GVL.pm[9].inConv.belt[0].fbconverter.freq <-> Axis#4 Outputs/Axis4 Frequency set through communication
//     PlcTask Outputs/GVL.pm[9].inConv.belt[1].fbconverter.freq <-> Axis#5 Outputs/Axis5 Frequency set through communication
//     PlcTask Outputs/GVL.pm[9].inConv.belt[2].fbconverter.freq <-> Axis#6 Outputs/Axis6 Frequency set through communication
//   kittingDeca/kittingDeca Instance <-> pm side/pm8_9_outerConv
//     PlcTask Inputs/GVL.pm[8].outConv.belt[0].fbconverter.running_freq <-> Axis#1 Iutputs/Axis1 Running frequency
//     PlcTask Inputs/GVL.pm[8].outConv.belt[1].fbconverter.running_freq <-> Axis#2 Iutputs/Axis2 Running frequency
//     PlcTask Inputs/GVL.pm[9].outConv.belt[0].fbconverter.running_freq <-> Axis#3 Iutputs/Axis3 Running frequency
//     PlcTask Inputs/GVL.pm[9].outConv.belt[1].fbconverter.running_freq <-> Axis#4 Iutputs/Axis4 Running frequency
//     PlcTask Inputs/GVL.pm[8].outConv.belt[0].fbconverter.status <-> Axis#1 Iutputs/Axis1 AC drive running status word 2
//     PlcTask Inputs/GVL.pm[8].outConv.belt[1].fbconverter.status <-> Axis#2 Iutputs/Axis2 AC drive running status word 2
//     PlcTask Inputs/GVL.pm[9].outConv.belt[0].fbconverter.status <-> Axis#3 Iutputs/Axis3 AC drive running status word 2
//     PlcTask Inputs/GVL.pm[9].outConv.belt[1].fbconverter.status <-> Axis#4 Iutputs/Axis4 AC drive running status word 2
//     PlcTask Outputs/GVL.pm[8].outConv.belt[0].fbconverter.cmd <-> Axis#1 Outputs/Axis1 Communication control command
//     PlcTask Outputs/GVL.pm[8].outConv.belt[1].fbconverter.cmd <-> Axis#2 Outputs/Axis2 Communication control command
//     PlcTask Outputs/GVL.pm[9].outConv.belt[0].fbconverter.cmd <-> Axis#3 Outputs/Axis3 Communication control command
//     PlcTask Outputs/GVL.pm[9].outConv.belt[1].fbconverter.cmd <-> Axis#4 Outputs/Axis4 Communication control command
//     PlcTask Outputs/GVL.pm[8].outConv.belt[0].fbconverter.freq <-> Axis#1 Outputs/Axis1 Frequency set through communication
//     PlcTask Outputs/GVL.pm[8].outConv.belt[1].fbconverter.freq <-> Axis#2 Outputs/Axis2 Frequency set through communication
//     PlcTask Outputs/GVL.pm[9].outConv.belt[0].fbconverter.freq <-> Axis#3 Outputs/Axis3 Frequency set through communication
//     PlcTask Outputs/GVL.pm[9].outConv.belt[1].fbconverter.freq <-> Axis#4 Outputs/Axis4 Frequency set through communication
//   kittingDeca/kittingDeca Instance <-> rem_wf/mcp_dio
//     PlcTask Inputs/G_IO.arDI[95]/Ch[0] <-> Module 1 (GL20-1600END)/1600END input-bit maping/Digital input CH1-bit0
//     PlcTask Inputs/G_IO.arDI[95]/Ch[10] <-> Module 1 (GL20-1600END)/1600END input-bit maping/Digital input CH2-bit2
//     PlcTask Inputs/G_IO.arDI[95]/Ch[11] <-> Module 1 (GL20-1600END)/1600END input-bit maping/Digital input CH2-bit3
//     PlcTask Inputs/G_IO.arDI[95]/Ch[12] <-> Module 1 (GL20-1600END)/1600END input-bit maping/Digital input CH2-bit4
//     PlcTask Inputs/G_IO.arDI[95]/Ch[13] <-> Module 1 (GL20-1600END)/1600END input-bit maping/Digital input CH2-bit5
//     PlcTask Inputs/G_IO.arDI[95]/Ch[14] <-> Module 1 (GL20-1600END)/1600END input-bit maping/Digital input CH2-bit6
//     PlcTask Inputs/G_IO.arDI[95]/Ch[15] <-> Module 1 (GL20-1600END)/1600END input-bit maping/Digital input CH2-bit7
//     PlcTask Inputs/G_IO.arDI[95]/Ch[1] <-> Module 1 (GL20-1600END)/1600END input-bit maping/Digital input CH1-bit1
//     PlcTask Inputs/G_IO.arDI[95]/Ch[2] <-> Module 1 (GL20-1600END)/1600END input-bit maping/Digital input CH1-bit2
//     PlcTask Inputs/G_IO.arDI[95]/Ch[3] <-> Module 1 (GL20-1600END)/1600END input-bit maping/Digital input CH1-bit3
//     PlcTask Inputs/G_IO.arDI[95]/Ch[4] <-> Module 1 (GL20-1600END)/1600END input-bit maping/Digital input CH1-bit4
//     PlcTask Inputs/G_IO.arDI[95]/Ch[5] <-> Module 1 (GL20-1600END)/1600END input-bit maping/Digital input CH1-bit5
//     PlcTask Inputs/G_IO.arDI[95]/Ch[6] <-> Module 1 (GL20-1600END)/1600END input-bit maping/Digital input CH1-bit6
//     PlcTask Inputs/G_IO.arDI[95]/Ch[7] <-> Module 1 (GL20-1600END)/1600END input-bit maping/Digital input CH1-bit7
//     PlcTask Inputs/G_IO.arDI[95]/Ch[8] <-> Module 1 (GL20-1600END)/1600END input-bit maping/Digital input CH2-bit0
//     PlcTask Inputs/G_IO.arDI[95]/Ch[9] <-> Module 1 (GL20-1600END)/1600END input-bit maping/Digital input CH2-bit1
//     PlcTask Outputs/G_IO.arDO[95]/Ch[0] <-> Module 2 (GL20-0016ETP)/0016ETP Output-bit maping/Digital output CH1-bit0
//     PlcTask Outputs/G_IO.arDO[95]/Ch[10] <-> Module 2 (GL20-0016ETP)/0016ETP Output-bit maping/Digital output CH2-bit2
//     PlcTask Outputs/G_IO.arDO[95]/Ch[11] <-> Module 2 (GL20-0016ETP)/0016ETP Output-bit maping/Digital output CH2-bit3
//     PlcTask Outputs/G_IO.arDO[95]/Ch[12] <-> Module 2 (GL20-0016ETP)/0016ETP Output-bit maping/Digital output CH2-bit4
//     PlcTask Outputs/G_IO.arDO[95]/Ch[13] <-> Module 2 (GL20-0016ETP)/0016ETP Output-bit maping/Digital output CH2-bit5
//     PlcTask Outputs/G_IO.arDO[95]/Ch[14] <-> Module 2 (GL20-0016ETP)/0016ETP Output-bit maping/Digital output CH2-bit6
//     PlcTask Outputs/G_IO.arDO[95]/Ch[15] <-> Module 2 (GL20-0016ETP)/0016ETP Output-bit maping/Digital output CH2-bit7
//     PlcTask Outputs/G_IO.arDO[95]/Ch[1] <-> Module 2 (GL20-0016ETP)/0016ETP Output-bit maping/Digital output CH1-bit1
//     PlcTask Outputs/G_IO.arDO[95]/Ch[2] <-> Module 2 (GL20-0016ETP)/0016ETP Output-bit maping/Digital output CH1-bit2
//     PlcTask Outputs/G_IO.arDO[95]/Ch[3] <-> Module 2 (GL20-0016ETP)/0016ETP Output-bit maping/Digital output CH1-bit3
//     PlcTask Outputs/G_IO.arDO[95]/Ch[4] <-> Module 2 (GL20-0016ETP)/0016ETP Output-bit maping/Digital output CH1-bit4
//     PlcTask Outputs/G_IO.arDO[95]/Ch[5] <-> Module 2 (GL20-0016ETP)/0016ETP Output-bit maping/Digital output CH1-bit5
//     PlcTask Outputs/G_IO.arDO[95]/Ch[6] <-> Module 2 (GL20-0016ETP)/0016ETP Output-bit maping/Digital output CH1-bit6
//     PlcTask Outputs/G_IO.arDO[95]/Ch[7] <-> Module 2 (GL20-0016ETP)/0016ETP Output-bit maping/Digital output CH1-bit7
//     PlcTask Outputs/G_IO.arDO[95]/Ch[8] <-> Module 2 (GL20-0016ETP)/0016ETP Output-bit maping/Digital output CH2-bit0
//     PlcTask Outputs/G_IO.arDO[95]/Ch[9] <-> Module 2 (GL20-0016ETP)/0016ETP Output-bit maping/Digital output CH2-bit1
//   kittingDeca/kittingDeca Instance <-> rem_wf/rem0_dio
//     PlcTask Inputs/G_IO.arDI[0]/Ch[0] <-> DI0/1600END input-bit maping/Digital input CH1-bit0
//     PlcTask Inputs/G_IO.arDI[0]/Ch[10] <-> DI0/1600END input-bit maping/Digital input CH2-bit2
//     PlcTask Inputs/G_IO.arDI[0]/Ch[11] <-> DI0/1600END input-bit maping/Digital input CH2-bit3
//     PlcTask Inputs/G_IO.arDI[0]/Ch[12] <-> DI0/1600END input-bit maping/Digital input CH2-bit4
//     PlcTask Inputs/G_IO.arDI[0]/Ch[13] <-> DI0/1600END input-bit maping/Digital input CH2-bit5
//     PlcTask Inputs/G_IO.arDI[0]/Ch[14] <-> DI0/1600END input-bit maping/Digital input CH2-bit6
//     PlcTask Inputs/G_IO.arDI[0]/Ch[15] <-> DI0/1600END input-bit maping/Digital input CH2-bit7
//     PlcTask Inputs/G_IO.arDI[0]/Ch[1] <-> DI0/1600END input-bit maping/Digital input CH1-bit1
//     PlcTask Inputs/G_IO.arDI[0]/Ch[2] <-> DI0/1600END input-bit maping/Digital input CH1-bit2
//     PlcTask Inputs/G_IO.arDI[0]/Ch[3] <-> DI0/1600END input-bit maping/Digital input CH1-bit3
//     PlcTask Inputs/G_IO.arDI[0]/Ch[4] <-> DI0/1600END input-bit maping/Digital input CH1-bit4
//     PlcTask Inputs/G_IO.arDI[0]/Ch[5] <-> DI0/1600END input-bit maping/Digital input CH1-bit5
//     PlcTask Inputs/G_IO.arDI[0]/Ch[6] <-> DI0/1600END input-bit maping/Digital input CH1-bit6
//     PlcTask Inputs/G_IO.arDI[0]/Ch[7] <-> DI0/1600END input-bit maping/Digital input CH1-bit7
//     PlcTask Inputs/G_IO.arDI[0]/Ch[8] <-> DI0/1600END input-bit maping/Digital input CH2-bit0
//     PlcTask Inputs/G_IO.arDI[0]/Ch[9] <-> DI0/1600END input-bit maping/Digital input CH2-bit1
//     PlcTask Inputs/G_IO.arDI[1]/Ch[0] <-> DI1/1600END input-bit maping/Digital input CH1-bit0
//     PlcTask Inputs/G_IO.arDI[1]/Ch[10] <-> DI1/1600END input-bit maping/Digital input CH2-bit2
//     PlcTask Inputs/G_IO.arDI[1]/Ch[11] <-> DI1/1600END input-bit maping/Digital input CH2-bit3
//     PlcTask Inputs/G_IO.arDI[1]/Ch[12] <-> DI1/1600END input-bit maping/Digital input CH2-bit4
//     PlcTask Inputs/G_IO.arDI[1]/Ch[13] <-> DI1/1600END input-bit maping/Digital input CH2-bit5
//     PlcTask Inputs/G_IO.arDI[1]/Ch[14] <-> DI1/1600END input-bit maping/Digital input CH2-bit6
//     PlcTask Inputs/G_IO.arDI[1]/Ch[15] <-> DI1/1600END input-bit maping/Digital input CH2-bit7
//     PlcTask Inputs/G_IO.arDI[1]/Ch[1] <-> DI1/1600END input-bit maping/Digital input CH1-bit1
//     PlcTask Inputs/G_IO.arDI[1]/Ch[2] <-> DI1/1600END input-bit maping/Digital input CH1-bit2
//     PlcTask Inputs/G_IO.arDI[1]/Ch[3] <-> DI1/1600END input-bit maping/Digital input CH1-bit3
//     PlcTask Inputs/G_IO.arDI[1]/Ch[4] <-> DI1/1600END input-bit maping/Digital input CH1-bit4
//     PlcTask Inputs/G_IO.arDI[1]/Ch[5] <-> DI1/1600END input-bit maping/Digital input CH1-bit5
//     PlcTask Inputs/G_IO.arDI[1]/Ch[6] <-> DI1/1600END input-bit maping/Digital input CH1-bit6
//     PlcTask Inputs/G_IO.arDI[1]/Ch[7] <-> DI1/1600END input-bit maping/Digital input CH1-bit7
//     PlcTask Inputs/G_IO.arDI[1]/Ch[8] <-> DI1/1600END input-bit maping/Digital input CH2-bit0
//     PlcTask Inputs/G_IO.arDI[1]/Ch[9] <-> DI1/1600END input-bit maping/Digital input CH2-bit1
//     PlcTask Inputs/G_IO.arDI[2]/Ch[0] <-> DI2/1600END input-bit maping/Digital input CH1-bit0
//     PlcTask Inputs/G_IO.arDI[2]/Ch[10] <-> DI2/1600END input-bit maping/Digital input CH2-bit2
//     PlcTask Inputs/G_IO.arDI[2]/Ch[11] <-> DI2/1600END input-bit maping/Digital input CH2-bit3
//     PlcTask Inputs/G_IO.arDI[2]/Ch[12] <-> DI2/1600END input-bit maping/Digital input CH2-bit4
//     PlcTask Inputs/G_IO.arDI[2]/Ch[13] <-> DI2/1600END input-bit maping/Digital input CH2-bit5
//     PlcTask Inputs/G_IO.arDI[2]/Ch[14] <-> DI2/1600END input-bit maping/Digital input CH2-bit6
//     PlcTask Inputs/G_IO.arDI[2]/Ch[15] <-> DI2/1600END input-bit maping/Digital input CH2-bit7
//     PlcTask Inputs/G_IO.arDI[2]/Ch[1] <-> DI2/1600END input-bit maping/Digital input CH1-bit1
//     PlcTask Inputs/G_IO.arDI[2]/Ch[2] <-> DI2/1600END input-bit maping/Digital input CH1-bit2
//     PlcTask Inputs/G_IO.arDI[2]/Ch[3] <-> DI2/1600END input-bit maping/Digital input CH1-bit3
//     PlcTask Inputs/G_IO.arDI[2]/Ch[4] <-> DI2/1600END input-bit maping/Digital input CH1-bit4
//     PlcTask Inputs/G_IO.arDI[2]/Ch[5] <-> DI2/1600END input-bit maping/Digital input CH1-bit5
//     PlcTask Inputs/G_IO.arDI[2]/Ch[6] <-> DI2/1600END input-bit maping/Digital input CH1-bit6
//     PlcTask Inputs/G_IO.arDI[2]/Ch[7] <-> DI2/1600END input-bit maping/Digital input CH1-bit7
//     PlcTask Inputs/G_IO.arDI[2]/Ch[8] <-> DI2/1600END input-bit maping/Digital input CH2-bit0
//     PlcTask Inputs/G_IO.arDI[2]/Ch[9] <-> DI2/1600END input-bit maping/Digital input CH2-bit1
//     PlcTask Inputs/G_IO.arDI[3]/Ch[0] <-> DI3/1600END input-bit maping/Digital input CH1-bit0
//     PlcTask Inputs/G_IO.arDI[3]/Ch[10] <-> DI3/1600END input-bit maping/Digital input CH2-bit2
//     PlcTask Inputs/G_IO.arDI[3]/Ch[11] <-> DI3/1600END input-bit maping/Digital input CH2-bit3
//     PlcTask Inputs/G_IO.arDI[3]/Ch[12] <-> DI3/1600END input-bit maping/Digital input CH2-bit4
//     PlcTask Inputs/G_IO.arDI[3]/Ch[13] <-> DI3/1600END input-bit maping/Digital input CH2-bit5
//     PlcTask Inputs/G_IO.arDI[3]/Ch[14] <-> DI3/1600END input-bit maping/Digital input CH2-bit6
//     PlcTask Inputs/G_IO.arDI[3]/Ch[15] <-> DI3/1600END input-bit maping/Digital input CH2-bit7
//     PlcTask Inputs/G_IO.arDI[3]/Ch[1] <-> DI3/1600END input-bit maping/Digital input CH1-bit1
//     PlcTask Inputs/G_IO.arDI[3]/Ch[2] <-> DI3/1600END input-bit maping/Digital input CH1-bit2
//     PlcTask Inputs/G_IO.arDI[3]/Ch[3] <-> DI3/1600END input-bit maping/Digital input CH1-bit3
//     PlcTask Inputs/G_IO.arDI[3]/Ch[4] <-> DI3/1600END input-bit maping/Digital input CH1-bit4
//     PlcTask Inputs/G_IO.arDI[3]/Ch[5] <-> DI3/1600END input-bit maping/Digital input CH1-bit5
//     PlcTask Inputs/G_IO.arDI[3]/Ch[6] <-> DI3/1600END input-bit maping/Digital input CH1-bit6
//     PlcTask Inputs/G_IO.arDI[3]/Ch[7] <-> DI3/1600END input-bit maping/Digital input CH1-bit7
//     PlcTask Inputs/G_IO.arDI[3]/Ch[8] <-> DI3/1600END input-bit maping/Digital input CH2-bit0
//     PlcTask Inputs/G_IO.arDI[3]/Ch[9] <-> DI3/1600END input-bit maping/Digital input CH2-bit1
//     PlcTask Outputs/G_IO.arDO[0]/Ch[0] <-> DO0/0016ETP Output-bit maping/Digital output CH1-bit0
//     PlcTask Outputs/G_IO.arDO[0]/Ch[10] <-> DO0/0016ETP Output-bit maping/Digital output CH2-bit2
//     PlcTask Outputs/G_IO.arDO[0]/Ch[11] <-> DO0/0016ETP Output-bit maping/Digital output CH2-bit3
//     PlcTask Outputs/G_IO.arDO[0]/Ch[12] <-> DO0/0016ETP Output-bit maping/Digital output CH2-bit4
//     PlcTask Outputs/G_IO.arDO[0]/Ch[13] <-> DO0/0016ETP Output-bit maping/Digital output CH2-bit5
//     PlcTask Outputs/G_IO.arDO[0]/Ch[14] <-> DO0/0016ETP Output-bit maping/Digital output CH2-bit6
//     PlcTask Outputs/G_IO.arDO[0]/Ch[15] <-> DO0/0016ETP Output-bit maping/Digital output CH2-bit7
//     PlcTask Outputs/G_IO.arDO[0]/Ch[1] <-> DO0/0016ETP Output-bit maping/Digital output CH1-bit1
//     PlcTask Outputs/G_IO.arDO[0]/Ch[2] <-> DO0/0016ETP Output-bit maping/Digital output CH1-bit2
//     PlcTask Outputs/G_IO.arDO[0]/Ch[3] <-> DO0/0016ETP Output-bit maping/Digital output CH1-bit3
//     PlcTask Outputs/G_IO.arDO[0]/Ch[4] <-> DO0/0016ETP Output-bit maping/Digital output CH1-bit4
//     PlcTask Outputs/G_IO.arDO[0]/Ch[5] <-> DO0/0016ETP Output-bit maping/Digital output CH1-bit5
//     PlcTask Outputs/G_IO.arDO[0]/Ch[6] <-> DO0/0016ETP Output-bit maping/Digital output CH1-bit6
//     PlcTask Outputs/G_IO.arDO[0]/Ch[7] <-> DO0/0016ETP Output-bit maping/Digital output CH1-bit7
//     PlcTask Outputs/G_IO.arDO[0]/Ch[8] <-> DO0/0016ETP Output-bit maping/Digital output CH2-bit0
//     PlcTask Outputs/G_IO.arDO[0]/Ch[9] <-> DO0/0016ETP Output-bit maping/Digital output CH2-bit1
//     PlcTask Outputs/G_IO.arDO[1]/Ch[0] <-> DO1/0016ETP Output-bit maping/Digital output CH1-bit0
//     PlcTask Outputs/G_IO.arDO[1]/Ch[10] <-> DO1/0016ETP Output-bit maping/Digital output CH2-bit2
//     PlcTask Outputs/G_IO.arDO[1]/Ch[11] <-> DO1/0016ETP Output-bit maping/Digital output CH2-bit3
//     PlcTask Outputs/G_IO.arDO[1]/Ch[12] <-> DO1/0016ETP Output-bit maping/Digital output CH2-bit4
//     PlcTask Outputs/G_IO.arDO[1]/Ch[13] <-> DO1/0016ETP Output-bit maping/Digital output CH2-bit5
//     PlcTask Outputs/G_IO.arDO[1]/Ch[14] <-> DO1/0016ETP Output-bit maping/Digital output CH2-bit6
//     PlcTask Outputs/G_IO.arDO[1]/Ch[15] <-> DO1/0016ETP Output-bit maping/Digital output CH2-bit7
//     PlcTask Outputs/G_IO.arDO[1]/Ch[1] <-> DO1/0016ETP Output-bit maping/Digital output CH1-bit1
//     PlcTask Outputs/G_IO.arDO[1]/Ch[2] <-> DO1/0016ETP Output-bit maping/Digital output CH1-bit2
//     PlcTask Outputs/G_IO.arDO[1]/Ch[3] <-> DO1/0016ETP Output-bit maping/Digital output CH1-bit3
//     PlcTask Outputs/G_IO.arDO[1]/Ch[4] <-> DO1/0016ETP Output-bit maping/Digital output CH1-bit4
//     PlcTask Outputs/G_IO.arDO[1]/Ch[5] <-> DO1/0016ETP Output-bit maping/Digital output CH1-bit5
//     PlcTask Outputs/G_IO.arDO[1]/Ch[6] <-> DO1/0016ETP Output-bit maping/Digital output CH1-bit6
//     PlcTask Outputs/G_IO.arDO[1]/Ch[7] <-> DO1/0016ETP Output-bit maping/Digital output CH1-bit7
//     PlcTask Outputs/G_IO.arDO[1]/Ch[8] <-> DO1/0016ETP Output-bit maping/Digital output CH2-bit0
//     PlcTask Outputs/G_IO.arDO[1]/Ch[9] <-> DO1/0016ETP Output-bit maping/Digital output CH2-bit1
//   kittingDeca/kittingDeca Instance <-> rem_wf/rem0_valve
//     PlcTask Outputs/G_IO.arDO[2]/Ch[0] <-> Module 1 (C2S-EC-24B)/Outputs/valve[1..4][0]
//     PlcTask Outputs/G_IO.arDO[2]/Ch[10] <-> Module 1 (C2S-EC-24B)/Outputs/valve[5..8][2]
//     PlcTask Outputs/G_IO.arDO[2]/Ch[11] <-> Module 1 (C2S-EC-24B)/Outputs/valve[5..8][3]
//     PlcTask Outputs/G_IO.arDO[2]/Ch[12] <-> Module 1 (C2S-EC-24B)/Outputs/valve[5..8][4]
//     PlcTask Outputs/G_IO.arDO[2]/Ch[13] <-> Module 1 (C2S-EC-24B)/Outputs/valve[5..8][5]
//     PlcTask Outputs/G_IO.arDO[2]/Ch[14] <-> Module 1 (C2S-EC-24B)/Outputs/valve[5..8][6]
//     PlcTask Outputs/G_IO.arDO[2]/Ch[15] <-> Module 1 (C2S-EC-24B)/Outputs/valve[5..8][7]
//     PlcTask Outputs/G_IO.arDO[2]/Ch[1] <-> Module 1 (C2S-EC-24B)/Outputs/valve[1..4][1]
//     PlcTask Outputs/G_IO.arDO[2]/Ch[2] <-> Module 1 (C2S-EC-24B)/Outputs/valve[1..4][2]
//     PlcTask Outputs/G_IO.arDO[2]/Ch[3] <-> Module 1 (C2S-EC-24B)/Outputs/valve[1..4][3]
//     PlcTask Outputs/G_IO.arDO[2]/Ch[4] <-> Module 1 (C2S-EC-24B)/Outputs/valve[1..4][4]
//     PlcTask Outputs/G_IO.arDO[2]/Ch[5] <-> Module 1 (C2S-EC-24B)/Outputs/valve[1..4][5]
//     PlcTask Outputs/G_IO.arDO[2]/Ch[6] <-> Module 1 (C2S-EC-24B)/Outputs/valve[1..4][6]
//     PlcTask Outputs/G_IO.arDO[2]/Ch[7] <-> Module 1 (C2S-EC-24B)/Outputs/valve[1..4][7]
//     PlcTask Outputs/G_IO.arDO[2]/Ch[8] <-> Module 1 (C2S-EC-24B)/Outputs/valve[5..8][0]
//     PlcTask Outputs/G_IO.arDO[2]/Ch[9] <-> Module 1 (C2S-EC-24B)/Outputs/valve[5..8][1]
//     PlcTask Outputs/G_IO.arDO[3]/Ch[0] <-> Module 1 (C2S-EC-24B)/Outputs/valve[9..12][0]
//     PlcTask Outputs/G_IO.arDO[3]/Ch[1] <-> Module 1 (C2S-EC-24B)/Outputs/valve[9..12][1]
//     PlcTask Outputs/G_IO.arDO[3]/Ch[2] <-> Module 1 (C2S-EC-24B)/Outputs/valve[9..12][2]
//     PlcTask Outputs/G_IO.arDO[3]/Ch[3] <-> Module 1 (C2S-EC-24B)/Outputs/valve[9..12][3]
//     PlcTask Outputs/G_IO.arDO[3]/Ch[4] <-> Module 1 (C2S-EC-24B)/Outputs/valve[9..12][4]
//     PlcTask Outputs/G_IO.arDO[3]/Ch[5] <-> Module 1 (C2S-EC-24B)/Outputs/valve[9..12][5]
//     PlcTask Outputs/G_IO.arDO[3]/Ch[6] <-> Module 1 (C2S-EC-24B)/Outputs/valve[9..12][6]
//     PlcTask Outputs/G_IO.arDO[3]/Ch[7] <-> Module 1 (C2S-EC-24B)/Outputs/valve[9..12][7]
//   kittingDeca/kittingDeca Instance <-> rem_wf/rem1_dio
//     PlcTask Inputs/G_IO.arDI[4]/Ch[0] <-> DI4/1600END input-bit maping/Digital input CH1-bit0
//     PlcTask Inputs/G_IO.arDI[4]/Ch[10] <-> DI4/1600END input-bit maping/Digital input CH2-bit2
//     PlcTask Inputs/G_IO.arDI[4]/Ch[11] <-> DI4/1600END input-bit maping/Digital input CH2-bit3
//     PlcTask Inputs/G_IO.arDI[4]/Ch[12] <-> DI4/1600END input-bit maping/Digital input CH2-bit4
//     PlcTask Inputs/G_IO.arDI[4]/Ch[13] <-> DI4/1600END input-bit maping/Digital input CH2-bit5
//     PlcTask Inputs/G_IO.arDI[4]/Ch[14] <-> DI4/1600END input-bit maping/Digital input CH2-bit6
//     PlcTask Inputs/G_IO.arDI[4]/Ch[15] <-> DI4/1600END input-bit maping/Digital input CH2-bit7
//     PlcTask Inputs/G_IO.arDI[4]/Ch[1] <-> DI4/1600END input-bit maping/Digital input CH1-bit1
//     PlcTask Inputs/G_IO.arDI[4]/Ch[2] <-> DI4/1600END input-bit maping/Digital input CH1-bit2
//     PlcTask Inputs/G_IO.arDI[4]/Ch[3] <-> DI4/1600END input-bit maping/Digital input CH1-bit3
//     PlcTask Inputs/G_IO.arDI[4]/Ch[4] <-> DI4/1600END input-bit maping/Digital input CH1-bit4
//     PlcTask Inputs/G_IO.arDI[4]/Ch[5] <-> DI4/1600END input-bit maping/Digital input CH1-bit5
//     PlcTask Inputs/G_IO.arDI[4]/Ch[6] <-> DI4/1600END input-bit maping/Digital input CH1-bit6
//     PlcTask Inputs/G_IO.arDI[4]/Ch[7] <-> DI4/1600END input-bit maping/Digital input CH1-bit7
//     PlcTask Inputs/G_IO.arDI[4]/Ch[8] <-> DI4/1600END input-bit maping/Digital input CH2-bit0
//     PlcTask Inputs/G_IO.arDI[4]/Ch[9] <-> DI4/1600END input-bit maping/Digital input CH2-bit1
//     PlcTask Inputs/G_IO.arDI[5]/Ch[0] <-> DI5/1600END input-bit maping/Digital input CH1-bit0
//     PlcTask Inputs/G_IO.arDI[5]/Ch[10] <-> DI5/1600END input-bit maping/Digital input CH2-bit2
//     PlcTask Inputs/G_IO.arDI[5]/Ch[11] <-> DI5/1600END input-bit maping/Digital input CH2-bit3
//     PlcTask Inputs/G_IO.arDI[5]/Ch[12] <-> DI5/1600END input-bit maping/Digital input CH2-bit4
//     PlcTask Inputs/G_IO.arDI[5]/Ch[13] <-> DI5/1600END input-bit maping/Digital input CH2-bit5
//     PlcTask Inputs/G_IO.arDI[5]/Ch[14] <-> DI5/1600END input-bit maping/Digital input CH2-bit6
//     PlcTask Inputs/G_IO.arDI[5]/Ch[15] <-> DI5/1600END input-bit maping/Digital input CH2-bit7
//     PlcTask Inputs/G_IO.arDI[5]/Ch[1] <-> DI5/1600END input-bit maping/Digital input CH1-bit1
//     PlcTask Inputs/G_IO.arDI[5]/Ch[2] <-> DI5/1600END input-bit maping/Digital input CH1-bit2
//     PlcTask Inputs/G_IO.arDI[5]/Ch[3] <-> DI5/1600END input-bit maping/Digital input CH1-bit3
//     PlcTask Inputs/G_IO.arDI[5]/Ch[4] <-> DI5/1600END input-bit maping/Digital input CH1-bit4
//     PlcTask Inputs/G_IO.arDI[5]/Ch[5] <-> DI5/1600END input-bit maping/Digital input CH1-bit5
//     PlcTask Inputs/G_IO.arDI[5]/Ch[6] <-> DI5/1600END input-bit maping/Digital input CH1-bit6
//     PlcTask Inputs/G_IO.arDI[5]/Ch[7] <-> DI5/1600END input-bit maping/Digital input CH1-bit7
//     PlcTask Inputs/G_IO.arDI[5]/Ch[8] <-> DI5/1600END input-bit maping/Digital input CH2-bit0
//     PlcTask Inputs/G_IO.arDI[5]/Ch[9] <-> DI5/1600END input-bit maping/Digital input CH2-bit1
//     PlcTask Inputs/G_IO.arDI[6]/Ch[0] <-> DI6/1600END input-bit maping/Digital input CH1-bit0
//     PlcTask Inputs/G_IO.arDI[6]/Ch[10] <-> DI6/1600END input-bit maping/Digital input CH2-bit2
//     PlcTask Inputs/G_IO.arDI[6]/Ch[11] <-> DI6/1600END input-bit maping/Digital input CH2-bit3
//     PlcTask Inputs/G_IO.arDI[6]/Ch[12] <-> DI6/1600END input-bit maping/Digital input CH2-bit4
//     PlcTask Inputs/G_IO.arDI[6]/Ch[13] <-> DI6/1600END input-bit maping/Digital input CH2-bit5
//     PlcTask Inputs/G_IO.arDI[6]/Ch[14] <-> DI6/1600END input-bit maping/Digital input CH2-bit6
//     PlcTask Inputs/G_IO.arDI[6]/Ch[15] <-> DI6/1600END input-bit maping/Digital input CH2-bit7
//     PlcTask Inputs/G_IO.arDI[6]/Ch[1] <-> DI6/1600END input-bit maping/Digital input CH1-bit1
//     PlcTask Inputs/G_IO.arDI[6]/Ch[2] <-> DI6/1600END input-bit maping/Digital input CH1-bit2
//     PlcTask Inputs/G_IO.arDI[6]/Ch[3] <-> DI6/1600END input-bit maping/Digital input CH1-bit3
//     PlcTask Inputs/G_IO.arDI[6]/Ch[4] <-> DI6/1600END input-bit maping/Digital input CH1-bit4
//     PlcTask Inputs/G_IO.arDI[6]/Ch[5] <-> DI6/1600END input-bit maping/Digital input CH1-bit5
//     PlcTask Inputs/G_IO.arDI[6]/Ch[6] <-> DI6/1600END input-bit maping/Digital input CH1-bit6
//     PlcTask Inputs/G_IO.arDI[6]/Ch[7] <-> DI6/1600END input-bit maping/Digital input CH1-bit7
//     PlcTask Inputs/G_IO.arDI[6]/Ch[8] <-> DI6/1600END input-bit maping/Digital input CH2-bit0
//     PlcTask Inputs/G_IO.arDI[6]/Ch[9] <-> DI6/1600END input-bit maping/Digital input CH2-bit1
//     PlcTask Inputs/G_IO.arDI[7]/Ch[0] <-> DI7/1600END input-bit maping/Digital input CH1-bit0
//     PlcTask Inputs/G_IO.arDI[7]/Ch[10] <-> DI7/1600END input-bit maping/Digital input CH2-bit2
//     PlcTask Inputs/G_IO.arDI[7]/Ch[11] <-> DI7/1600END input-bit maping/Digital input CH2-bit3
//     PlcTask Inputs/G_IO.arDI[7]/Ch[12] <-> DI7/1600END input-bit maping/Digital input CH2-bit4
//     PlcTask Inputs/G_IO.arDI[7]/Ch[13] <-> DI7/1600END input-bit maping/Digital input CH2-bit5
//     PlcTask Inputs/G_IO.arDI[7]/Ch[14] <-> DI7/1600END input-bit maping/Digital input CH2-bit6
//     PlcTask Inputs/G_IO.arDI[7]/Ch[15] <-> DI7/1600END input-bit maping/Digital input CH2-bit7
//     PlcTask Inputs/G_IO.arDI[7]/Ch[1] <-> DI7/1600END input-bit maping/Digital input CH1-bit1
//     PlcTask Inputs/G_IO.arDI[7]/Ch[2] <-> DI7/1600END input-bit maping/Digital input CH1-bit2
//     PlcTask Inputs/G_IO.arDI[7]/Ch[3] <-> DI7/1600END input-bit maping/Digital input CH1-bit3
//     PlcTask Inputs/G_IO.arDI[7]/Ch[4] <-> DI7/1600END input-bit maping/Digital input CH1-bit4
//     PlcTask Inputs/G_IO.arDI[7]/Ch[5] <-> DI7/1600END input-bit maping/Digital input CH1-bit5
//     PlcTask Inputs/G_IO.arDI[7]/Ch[6] <-> DI7/1600END input-bit maping/Digital input CH1-bit6
//     PlcTask Inputs/G_IO.arDI[7]/Ch[7] <-> DI7/1600END input-bit maping/Digital input CH1-bit7
//     PlcTask Inputs/G_IO.arDI[7]/Ch[8] <-> DI7/1600END input-bit maping/Digital input CH2-bit0
//     PlcTask Inputs/G_IO.arDI[7]/Ch[9] <-> DI7/1600END input-bit maping/Digital input CH2-bit1
//     PlcTask Outputs/G_IO.arDO[4]/Ch[0] <-> DO4/0016ETP Output-bit maping/Digital output CH1-bit0
//     PlcTask Outputs/G_IO.arDO[4]/Ch[10] <-> DO4/0016ETP Output-bit maping/Digital output CH2-bit2
//     PlcTask Outputs/G_IO.arDO[4]/Ch[11] <-> DO4/0016ETP Output-bit maping/Digital output CH2-bit3
//     PlcTask Outputs/G_IO.arDO[4]/Ch[12] <-> DO4/0016ETP Output-bit maping/Digital output CH2-bit4
//     PlcTask Outputs/G_IO.arDO[4]/Ch[13] <-> DO4/0016ETP Output-bit maping/Digital output CH2-bit5
//     PlcTask Outputs/G_IO.arDO[4]/Ch[14] <-> DO4/0016ETP Output-bit maping/Digital output CH2-bit6
//     PlcTask Outputs/G_IO.arDO[4]/Ch[15] <-> DO4/0016ETP Output-bit maping/Digital output CH2-bit7
//     PlcTask Outputs/G_IO.arDO[4]/Ch[1] <-> DO4/0016ETP Output-bit maping/Digital output CH1-bit1
//     PlcTask Outputs/G_IO.arDO[4]/Ch[2] <-> DO4/0016ETP Output-bit maping/Digital output CH1-bit2
//     PlcTask Outputs/G_IO.arDO[4]/Ch[3] <-> DO4/0016ETP Output-bit maping/Digital output CH1-bit3
//     PlcTask Outputs/G_IO.arDO[4]/Ch[4] <-> DO4/0016ETP Output-bit maping/Digital output CH1-bit4
//     PlcTask Outputs/G_IO.arDO[4]/Ch[5] <-> DO4/0016ETP Output-bit maping/Digital output CH1-bit5
//     PlcTask Outputs/G_IO.arDO[4]/Ch[6] <-> DO4/0016ETP Output-bit maping/Digital output CH1-bit6
//     PlcTask Outputs/G_IO.arDO[4]/Ch[7] <-> DO4/0016ETP Output-bit maping/Digital output CH1-bit7
//     PlcTask Outputs/G_IO.arDO[4]/Ch[8] <-> DO4/0016ETP Output-bit maping/Digital output CH2-bit0
//     PlcTask Outputs/G_IO.arDO[4]/Ch[9] <-> DO4/0016ETP Output-bit maping/Digital output CH2-bit1
//     PlcTask Outputs/G_IO.arDO[5]/Ch[0] <-> DO5/0016ETP Output-bit maping/Digital output CH1-bit0
//     PlcTask Outputs/G_IO.arDO[5]/Ch[10] <-> DO5/0016ETP Output-bit maping/Digital output CH2-bit2
//     PlcTask Outputs/G_IO.arDO[5]/Ch[11] <-> DO5/0016ETP Output-bit maping/Digital output CH2-bit3
//     PlcTask Outputs/G_IO.arDO[5]/Ch[12] <-> DO5/0016ETP Output-bit maping/Digital output CH2-bit4
//     PlcTask Outputs/G_IO.arDO[5]/Ch[13] <-> DO5/0016ETP Output-bit maping/Digital output CH2-bit5
//     PlcTask Outputs/G_IO.arDO[5]/Ch[14] <-> DO5/0016ETP Output-bit maping/Digital output CH2-bit6
//     PlcTask Outputs/G_IO.arDO[5]/Ch[15] <-> DO5/0016ETP Output-bit maping/Digital output CH2-bit7
//     PlcTask Outputs/G_IO.arDO[5]/Ch[1] <-> DO5/0016ETP Output-bit maping/Digital output CH1-bit1
//     PlcTask Outputs/G_IO.arDO[5]/Ch[2] <-> DO5/0016ETP Output-bit maping/Digital output CH1-bit2
//     PlcTask Outputs/G_IO.arDO[5]/Ch[3] <-> DO5/0016ETP Output-bit maping/Digital output CH1-bit3
//     PlcTask Outputs/G_IO.arDO[5]/Ch[4] <-> DO5/0016ETP Output-bit maping/Digital output CH1-bit4
//     PlcTask Outputs/G_IO.arDO[5]/Ch[5] <-> DO5/0016ETP Output-bit maping/Digital output CH1-bit5
//     PlcTask Outputs/G_IO.arDO[5]/Ch[6] <-> DO5/0016ETP Output-bit maping/Digital output CH1-bit6
//     PlcTask Outputs/G_IO.arDO[5]/Ch[7] <-> DO5/0016ETP Output-bit maping/Digital output CH1-bit7
//     PlcTask Outputs/G_IO.arDO[5]/Ch[8] <-> DO5/0016ETP Output-bit maping/Digital output CH2-bit0
//     PlcTask Outputs/G_IO.arDO[5]/Ch[9] <-> DO5/0016ETP Output-bit maping/Digital output CH2-bit1
//   kittingDeca/kittingDeca Instance <-> rem_wf/rem1_valve
//     PlcTask Outputs/G_IO.arDO[6]/Ch[0] <-> Module 1 (C2S-EC-24B)/Outputs/valve[1..4][0]
//     PlcTask Outputs/G_IO.arDO[6]/Ch[10] <-> Module 1 (C2S-EC-24B)/Outputs/valve[5..8][2]
//     PlcTask Outputs/G_IO.arDO[6]/Ch[11] <-> Module 1 (C2S-EC-24B)/Outputs/valve[5..8][3]
//     PlcTask Outputs/G_IO.arDO[6]/Ch[12] <-> Module 1 (C2S-EC-24B)/Outputs/valve[5..8][4]
//     PlcTask Outputs/G_IO.arDO[6]/Ch[13] <-> Module 1 (C2S-EC-24B)/Outputs/valve[5..8][5]
//     PlcTask Outputs/G_IO.arDO[6]/Ch[14] <-> Module 1 (C2S-EC-24B)/Outputs/valve[5..8][6]
//     PlcTask Outputs/G_IO.arDO[6]/Ch[15] <-> Module 1 (C2S-EC-24B)/Outputs/valve[5..8][7]
//     PlcTask Outputs/G_IO.arDO[6]/Ch[1] <-> Module 1 (C2S-EC-24B)/Outputs/valve[1..4][1]
//     PlcTask Outputs/G_IO.arDO[6]/Ch[2] <-> Module 1 (C2S-EC-24B)/Outputs/valve[1..4][2]
//     PlcTask Outputs/G_IO.arDO[6]/Ch[3] <-> Module 1 (C2S-EC-24B)/Outputs/valve[1..4][3]
//     PlcTask Outputs/G_IO.arDO[6]/Ch[4] <-> Module 1 (C2S-EC-24B)/Outputs/valve[1..4][4]
//     PlcTask Outputs/G_IO.arDO[6]/Ch[5] <-> Module 1 (C2S-EC-24B)/Outputs/valve[1..4][5]
//     PlcTask Outputs/G_IO.arDO[6]/Ch[6] <-> Module 1 (C2S-EC-24B)/Outputs/valve[1..4][6]
//     PlcTask Outputs/G_IO.arDO[6]/Ch[7] <-> Module 1 (C2S-EC-24B)/Outputs/valve[1..4][7]
//     PlcTask Outputs/G_IO.arDO[6]/Ch[8] <-> Module 1 (C2S-EC-24B)/Outputs/valve[5..8][0]
//     PlcTask Outputs/G_IO.arDO[6]/Ch[9] <-> Module 1 (C2S-EC-24B)/Outputs/valve[5..8][1]
//     PlcTask Outputs/G_IO.arDO[7]/Ch[0] <-> Module 1 (C2S-EC-24B)/Outputs/valve[9..12][0]
//     PlcTask Outputs/G_IO.arDO[7]/Ch[1] <-> Module 1 (C2S-EC-24B)/Outputs/valve[9..12][1]
//     PlcTask Outputs/G_IO.arDO[7]/Ch[2] <-> Module 1 (C2S-EC-24B)/Outputs/valve[9..12][2]
//     PlcTask Outputs/G_IO.arDO[7]/Ch[3] <-> Module 1 (C2S-EC-24B)/Outputs/valve[9..12][3]
//     PlcTask Outputs/G_IO.arDO[7]/Ch[4] <-> Module 1 (C2S-EC-24B)/Outputs/valve[9..12][4]
//     PlcTask Outputs/G_IO.arDO[7]/Ch[5] <-> Module 1 (C2S-EC-24B)/Outputs/valve[9..12][5]
//     PlcTask Outputs/G_IO.arDO[7]/Ch[6] <-> Module 1 (C2S-EC-24B)/Outputs/valve[9..12][6]
//     PlcTask Outputs/G_IO.arDO[7]/Ch[7] <-> Module 1 (C2S-EC-24B)/Outputs/valve[9..12][7]
//   kittingDeca/kittingDeca Instance <-> rem_wf/rem2_dio
//     PlcTask Inputs/G_IO.arDI[10]/Ch[0] <-> DI10/1600END input-bit maping/Digital input CH1-bit0
//     PlcTask Inputs/G_IO.arDI[10]/Ch[10] <-> DI10/1600END input-bit maping/Digital input CH2-bit2
//     PlcTask Inputs/G_IO.arDI[10]/Ch[11] <-> DI10/1600END input-bit maping/Digital input CH2-bit3
//     PlcTask Inputs/G_IO.arDI[10]/Ch[12] <-> DI10/1600END input-bit maping/Digital input CH2-bit4
//     PlcTask Inputs/G_IO.arDI[10]/Ch[13] <-> DI10/1600END input-bit maping/Digital input CH2-bit5
//     PlcTask Inputs/G_IO.arDI[10]/Ch[14] <-> DI10/1600END input-bit maping/Digital input CH2-bit6
//     PlcTask Inputs/G_IO.arDI[10]/Ch[15] <-> DI10/1600END input-bit maping/Digital input CH2-bit7
//     PlcTask Inputs/G_IO.arDI[10]/Ch[1] <-> DI10/1600END input-bit maping/Digital input CH1-bit1
//     PlcTask Inputs/G_IO.arDI[10]/Ch[2] <-> DI10/1600END input-bit maping/Digital input CH1-bit2
//     PlcTask Inputs/G_IO.arDI[10]/Ch[3] <-> DI10/1600END input-bit maping/Digital input CH1-bit3
//     PlcTask Inputs/G_IO.arDI[10]/Ch[4] <-> DI10/1600END input-bit maping/Digital input CH1-bit4
//     PlcTask Inputs/G_IO.arDI[10]/Ch[5] <-> DI10/1600END input-bit maping/Digital input CH1-bit5
//     PlcTask Inputs/G_IO.arDI[10]/Ch[6] <-> DI10/1600END input-bit maping/Digital input CH1-bit6
//     PlcTask Inputs/G_IO.arDI[10]/Ch[7] <-> DI10/1600END input-bit maping/Digital input CH1-bit7
//     PlcTask Inputs/G_IO.arDI[10]/Ch[8] <-> DI10/1600END input-bit maping/Digital input CH2-bit0
//     PlcTask Inputs/G_IO.arDI[10]/Ch[9] <-> DI10/1600END input-bit maping/Digital input CH2-bit1
//     PlcTask Inputs/G_IO.arDI[11]/Ch[0] <-> DI11/1600END input-bit maping/Digital input CH1-bit0
//     PlcTask Inputs/G_IO.arDI[11]/Ch[10] <-> DI11/1600END input-bit maping/Digital input CH2-bit2
//     PlcTask Inputs/G_IO.arDI[11]/Ch[11] <-> DI11/1600END input-bit maping/Digital input CH2-bit3
//     PlcTask Inputs/G_IO.arDI[11]/Ch[12] <-> DI11/1600END input-bit maping/Digital input CH2-bit4
//     PlcTask Inputs/G_IO.arDI[11]/Ch[13] <-> DI11/1600END input-bit maping/Digital input CH2-bit5
//     PlcTask Inputs/G_IO.arDI[11]/Ch[14] <-> DI11/1600END input-bit maping/Digital input CH2-bit6
//     PlcTask Inputs/G_IO.arDI[11]/Ch[15] <-> DI11/1600END input-bit maping/Digital input CH2-bit7
//     PlcTask Inputs/G_IO.arDI[11]/Ch[1] <-> DI11/1600END input-bit maping/Digital input CH1-bit1
//     PlcTask Inputs/G_IO.arDI[11]/Ch[2] <-> DI11/1600END input-bit maping/Digital input CH1-bit2
//     PlcTask Inputs/G_IO.arDI[11]/Ch[3] <-> DI11/1600END input-bit maping/Digital input CH1-bit3
//     PlcTask Inputs/G_IO.arDI[11]/Ch[4] <-> DI11/1600END input-bit maping/Digital input CH1-bit4
//     PlcTask Inputs/G_IO.arDI[11]/Ch[5] <-> DI11/1600END input-bit maping/Digital input CH1-bit5
//     PlcTask Inputs/G_IO.arDI[11]/Ch[6] <-> DI11/1600END input-bit maping/Digital input CH1-bit6
//     PlcTask Inputs/G_IO.arDI[11]/Ch[7] <-> DI11/1600END input-bit maping/Digital input CH1-bit7
//     PlcTask Inputs/G_IO.arDI[11]/Ch[8] <-> DI11/1600END input-bit maping/Digital input CH2-bit0
//     PlcTask Inputs/G_IO.arDI[11]/Ch[9] <-> DI11/1600END input-bit maping/Digital input CH2-bit1
//     PlcTask Inputs/G_IO.arDI[8]/Ch[0] <-> DI8/1600END input-bit maping/Digital input CH1-bit0
//     PlcTask Inputs/G_IO.arDI[8]/Ch[10] <-> DI8/1600END input-bit maping/Digital input CH2-bit2
//     PlcTask Inputs/G_IO.arDI[8]/Ch[11] <-> DI8/1600END input-bit maping/Digital input CH2-bit3
//     PlcTask Inputs/G_IO.arDI[8]/Ch[12] <-> DI8/1600END input-bit maping/Digital input CH2-bit4
//     PlcTask Inputs/G_IO.arDI[8]/Ch[13] <-> DI8/1600END input-bit maping/Digital input CH2-bit5
//     PlcTask Inputs/G_IO.arDI[8]/Ch[14] <-> DI8/1600END input-bit maping/Digital input CH2-bit6
//     PlcTask Inputs/G_IO.arDI[8]/Ch[15] <-> DI8/1600END input-bit maping/Digital input CH2-bit7
//     PlcTask Inputs/G_IO.arDI[8]/Ch[1] <-> DI8/1600END input-bit maping/Digital input CH1-bit1
//     PlcTask Inputs/G_IO.arDI[8]/Ch[2] <-> DI8/1600END input-bit maping/Digital input CH1-bit2
//     PlcTask Inputs/G_IO.arDI[8]/Ch[3] <-> DI8/1600END input-bit maping/Digital input CH1-bit3
//     PlcTask Inputs/G_IO.arDI[8]/Ch[4] <-> DI8/1600END input-bit maping/Digital input CH1-bit4
//     PlcTask Inputs/G_IO.arDI[8]/Ch[5] <-> DI8/1600END input-bit maping/Digital input CH1-bit5
//     PlcTask Inputs/G_IO.arDI[8]/Ch[6] <-> DI8/1600END input-bit maping/Digital input CH1-bit6
//     PlcTask Inputs/G_IO.arDI[8]/Ch[7] <-> DI8/1600END input-bit maping/Digital input CH1-bit7
//     PlcTask Inputs/G_IO.arDI[8]/Ch[8] <-> DI8/1600END input-bit maping/Digital input CH2-bit0
//     PlcTask Inputs/G_IO.arDI[8]/Ch[9] <-> DI8/1600END input-bit maping/Digital input CH2-bit1
//     PlcTask Inputs/G_IO.arDI[9]/Ch[0] <-> DI9/1600END input-bit maping/Digital input CH1-bit0
//     PlcTask Inputs/G_IO.arDI[9]/Ch[10] <-> DI9/1600END input-bit maping/Digital input CH2-bit2
//     PlcTask Inputs/G_IO.arDI[9]/Ch[11] <-> DI9/1600END input-bit maping/Digital input CH2-bit3
//     PlcTask Inputs/G_IO.arDI[9]/Ch[12] <-> DI9/1600END input-bit maping/Digital input CH2-bit4
//     PlcTask Inputs/G_IO.arDI[9]/Ch[13] <-> DI9/1600END input-bit maping/Digital input CH2-bit5
//     PlcTask Inputs/G_IO.arDI[9]/Ch[14] <-> DI9/1600END input-bit maping/Digital input CH2-bit6
//     PlcTask Inputs/G_IO.arDI[9]/Ch[15] <-> DI9/1600END input-bit maping/Digital input CH2-bit7
//     PlcTask Inputs/G_IO.arDI[9]/Ch[1] <-> DI9/1600END input-bit maping/Digital input CH1-bit1
//     PlcTask Inputs/G_IO.arDI[9]/Ch[2] <-> DI9/1600END input-bit maping/Digital input CH1-bit2
//     PlcTask Inputs/G_IO.arDI[9]/Ch[3] <-> DI9/1600END input-bit maping/Digital input CH1-bit3
//     PlcTask Inputs/G_IO.arDI[9]/Ch[4] <-> DI9/1600END input-bit maping/Digital input CH1-bit4
//     PlcTask Inputs/G_IO.arDI[9]/Ch[5] <-> DI9/1600END input-bit maping/Digital input CH1-bit5
//     PlcTask Inputs/G_IO.arDI[9]/Ch[6] <-> DI9/1600END input-bit maping/Digital input CH1-bit6
//     PlcTask Inputs/G_IO.arDI[9]/Ch[7] <-> DI9/1600END input-bit maping/Digital input CH1-bit7
//     PlcTask Inputs/G_IO.arDI[9]/Ch[8] <-> DI9/1600END input-bit maping/Digital input CH2-bit0
//     PlcTask Inputs/G_IO.arDI[9]/Ch[9] <-> DI9/1600END input-bit maping/Digital input CH2-bit1
//     PlcTask Outputs/G_IO.arDO[8]/Ch[0] <-> DO8/0016ETP Output-bit maping/Digital output CH1-bit0
//     PlcTask Outputs/G_IO.arDO[8]/Ch[10] <-> DO8/0016ETP Output-bit maping/Digital output CH2-bit2
//     PlcTask Outputs/G_IO.arDO[8]/Ch[11] <-> DO8/0016ETP Output-bit maping/Digital output CH2-bit3
//     PlcTask Outputs/G_IO.arDO[8]/Ch[12] <-> DO8/0016ETP Output-bit maping/Digital output CH2-bit4
//     PlcTask Outputs/G_IO.arDO[8]/Ch[13] <-> DO8/0016ETP Output-bit maping/Digital output CH2-bit5
//     PlcTask Outputs/G_IO.arDO[8]/Ch[14] <-> DO8/0016ETP Output-bit maping/Digital output CH2-bit6
//     PlcTask Outputs/G_IO.arDO[8]/Ch[15] <-> DO8/0016ETP Output-bit maping/Digital output CH2-bit7
//     PlcTask Outputs/G_IO.arDO[8]/Ch[1] <-> DO8/0016ETP Output-bit maping/Digital output CH1-bit1
//     PlcTask Outputs/G_IO.arDO[8]/Ch[2] <-> DO8/0016ETP Output-bit maping/Digital output CH1-bit2
//     PlcTask Outputs/G_IO.arDO[8]/Ch[3] <-> DO8/0016ETP Output-bit maping/Digital output CH1-bit3
//     PlcTask Outputs/G_IO.arDO[8]/Ch[4] <-> DO8/0016ETP Output-bit maping/Digital output CH1-bit4
//     PlcTask Outputs/G_IO.arDO[8]/Ch[5] <-> DO8/0016ETP Output-bit maping/Digital output CH1-bit5
//     PlcTask Outputs/G_IO.arDO[8]/Ch[6] <-> DO8/0016ETP Output-bit maping/Digital output CH1-bit6
//     PlcTask Outputs/G_IO.arDO[8]/Ch[7] <-> DO8/0016ETP Output-bit maping/Digital output CH1-bit7
//     PlcTask Outputs/G_IO.arDO[8]/Ch[8] <-> DO8/0016ETP Output-bit maping/Digital output CH2-bit0
//     PlcTask Outputs/G_IO.arDO[8]/Ch[9] <-> DO8/0016ETP Output-bit maping/Digital output CH2-bit1
//     PlcTask Outputs/G_IO.arDO[9]/Ch[0] <-> DO9/0016ETP Output-bit maping/Digital output CH1-bit0
//     PlcTask Outputs/G_IO.arDO[9]/Ch[10] <-> DO9/0016ETP Output-bit maping/Digital output CH2-bit2
//     PlcTask Outputs/G_IO.arDO[9]/Ch[11] <-> DO9/0016ETP Output-bit maping/Digital output CH2-bit3
//     PlcTask Outputs/G_IO.arDO[9]/Ch[12] <-> DO9/0016ETP Output-bit maping/Digital output CH2-bit4
//     PlcTask Outputs/G_IO.arDO[9]/Ch[13] <-> DO9/0016ETP Output-bit maping/Digital output CH2-bit5
//     PlcTask Outputs/G_IO.arDO[9]/Ch[14] <-> DO9/0016ETP Output-bit maping/Digital output CH2-bit6
//     PlcTask Outputs/G_IO.arDO[9]/Ch[15] <-> DO9/0016ETP Output-bit maping/Digital output CH2-bit7
//     PlcTask Outputs/G_IO.arDO[9]/Ch[1] <-> DO9/0016ETP Output-bit maping/Digital output CH1-bit1
//     PlcTask Outputs/G_IO.arDO[9]/Ch[2] <-> DO9/0016ETP Output-bit maping/Digital output CH1-bit2
//     PlcTask Outputs/G_IO.arDO[9]/Ch[3] <-> DO9/0016ETP Output-bit maping/Digital output CH1-bit3
//     PlcTask Outputs/G_IO.arDO[9]/Ch[4] <-> DO9/0016ETP Output-bit maping/Digital output CH1-bit4
//     PlcTask Outputs/G_IO.arDO[9]/Ch[5] <-> DO9/0016ETP Output-bit maping/Digital output CH1-bit5
//     PlcTask Outputs/G_IO.arDO[9]/Ch[6] <-> DO9/0016ETP Output-bit maping/Digital output CH1-bit6
//     PlcTask Outputs/G_IO.arDO[9]/Ch[7] <-> DO9/0016ETP Output-bit maping/Digital output CH1-bit7
//     PlcTask Outputs/G_IO.arDO[9]/Ch[8] <-> DO9/0016ETP Output-bit maping/Digital output CH2-bit0
//     PlcTask Outputs/G_IO.arDO[9]/Ch[9] <-> DO9/0016ETP Output-bit maping/Digital output CH2-bit1
//   kittingDeca/kittingDeca Instance <-> rem_wf/rem2_valve
//     PlcTask Outputs/G_IO.arDO[10]/Ch[0] <-> Module 1 (C2S-EC-24B)/Outputs/valve[1..4][0]
//     PlcTask Outputs/G_IO.arDO[10]/Ch[10] <-> Module 1 (C2S-EC-24B)/Outputs/valve[5..8][2]
//     PlcTask Outputs/G_IO.arDO[10]/Ch[11] <-> Module 1 (C2S-EC-24B)/Outputs/valve[5..8][3]
//     PlcTask Outputs/G_IO.arDO[10]/Ch[12] <-> Module 1 (C2S-EC-24B)/Outputs/valve[5..8][4]
//     PlcTask Outputs/G_IO.arDO[10]/Ch[13] <-> Module 1 (C2S-EC-24B)/Outputs/valve[5..8][5]
//     PlcTask Outputs/G_IO.arDO[10]/Ch[14] <-> Module 1 (C2S-EC-24B)/Outputs/valve[5..8][6]
//     PlcTask Outputs/G_IO.arDO[10]/Ch[15] <-> Module 1 (C2S-EC-24B)/Outputs/valve[5..8][7]
//     PlcTask Outputs/G_IO.arDO[10]/Ch[1] <-> Module 1 (C2S-EC-24B)/Outputs/valve[1..4][1]
//     PlcTask Outputs/G_IO.arDO[10]/Ch[2] <-> Module 1 (C2S-EC-24B)/Outputs/valve[1..4][2]
//     PlcTask Outputs/G_IO.arDO[10]/Ch[3] <-> Module 1 (C2S-EC-24B)/Outputs/valve[1..4][3]
//     PlcTask Outputs/G_IO.arDO[10]/Ch[4] <-> Module 1 (C2S-EC-24B)/Outputs/valve[1..4][4]
//     PlcTask Outputs/G_IO.arDO[10]/Ch[5] <-> Module 1 (C2S-EC-24B)/Outputs/valve[1..4][5]
//     PlcTask Outputs/G_IO.arDO[10]/Ch[6] <-> Module 1 (C2S-EC-24B)/Outputs/valve[1..4][6]
//     PlcTask Outputs/G_IO.arDO[10]/Ch[7] <-> Module 1 (C2S-EC-24B)/Outputs/valve[1..4][7]
//     PlcTask Outputs/G_IO.arDO[10]/Ch[8] <-> Module 1 (C2S-EC-24B)/Outputs/valve[5..8][0]
//     PlcTask Outputs/G_IO.arDO[10]/Ch[9] <-> Module 1 (C2S-EC-24B)/Outputs/valve[5..8][1]
//     PlcTask Outputs/G_IO.arDO[11]/Ch[0] <-> Module 1 (C2S-EC-24B)/Outputs/valve[9..12][0]
//     PlcTask Outputs/G_IO.arDO[11]/Ch[1] <-> Module 1 (C2S-EC-24B)/Outputs/valve[9..12][1]
//     PlcTask Outputs/G_IO.arDO[11]/Ch[2] <-> Module 1 (C2S-EC-24B)/Outputs/valve[9..12][2]
//     PlcTask Outputs/G_IO.arDO[11]/Ch[3] <-> Module 1 (C2S-EC-24B)/Outputs/valve[9..12][3]
//     PlcTask Outputs/G_IO.arDO[11]/Ch[4] <-> Module 1 (C2S-EC-24B)/Outputs/valve[9..12][4]
//     PlcTask Outputs/G_IO.arDO[11]/Ch[5] <-> Module 1 (C2S-EC-24B)/Outputs/valve[9..12][5]
//     PlcTask Outputs/G_IO.arDO[11]/Ch[6] <-> Module 1 (C2S-EC-24B)/Outputs/valve[9..12][6]
//     PlcTask Outputs/G_IO.arDO[11]/Ch[7] <-> Module 1 (C2S-EC-24B)/Outputs/valve[9..12][7]
//   kittingDeca/kittingDeca Instance <-> rem_wf/rem3_dio
//     PlcTask Inputs/G_IO.arDI[12]/Ch[0] <-> DI12/1600END input-bit maping/Digital input CH1-bit0
//     PlcTask Inputs/G_IO.arDI[12]/Ch[10] <-> DI12/1600END input-bit maping/Digital input CH2-bit2
//     PlcTask Inputs/G_IO.arDI[12]/Ch[11] <-> DI12/1600END input-bit maping/Digital input CH2-bit3
//     PlcTask Inputs/G_IO.arDI[12]/Ch[12] <-> DI12/1600END input-bit maping/Digital input CH2-bit4
//     PlcTask Inputs/G_IO.arDI[12]/Ch[13] <-> DI12/1600END input-bit maping/Digital input CH2-bit5
//     PlcTask Inputs/G_IO.arDI[12]/Ch[14] <-> DI12/1600END input-bit maping/Digital input CH2-bit6
//     PlcTask Inputs/G_IO.arDI[12]/Ch[15] <-> DI12/1600END input-bit maping/Digital input CH2-bit7
//     PlcTask Inputs/G_IO.arDI[12]/Ch[1] <-> DI12/1600END input-bit maping/Digital input CH1-bit1
//     PlcTask Inputs/G_IO.arDI[12]/Ch[2] <-> DI12/1600END input-bit maping/Digital input CH1-bit2
//     PlcTask Inputs/G_IO.arDI[12]/Ch[3] <-> DI12/1600END input-bit maping/Digital input CH1-bit3
//     PlcTask Inputs/G_IO.arDI[12]/Ch[4] <-> DI12/1600END input-bit maping/Digital input CH1-bit4
//     PlcTask Inputs/G_IO.arDI[12]/Ch[5] <-> DI12/1600END input-bit maping/Digital input CH1-bit5
//     PlcTask Inputs/G_IO.arDI[12]/Ch[6] <-> DI12/1600END input-bit maping/Digital input CH1-bit6
//     PlcTask Inputs/G_IO.arDI[12]/Ch[7] <-> DI12/1600END input-bit maping/Digital input CH1-bit7
//     PlcTask Inputs/G_IO.arDI[12]/Ch[8] <-> DI12/1600END input-bit maping/Digital input CH2-bit0
//     PlcTask Inputs/G_IO.arDI[12]/Ch[9] <-> DI12/1600END input-bit maping/Digital input CH2-bit1
//     PlcTask Inputs/G_IO.arDI[13]/Ch[0] <-> DI13/1600END input-bit maping/Digital input CH1-bit0
//     PlcTask Inputs/G_IO.arDI[13]/Ch[10] <-> DI13/1600END input-bit maping/Digital input CH2-bit2
//     PlcTask Inputs/G_IO.arDI[13]/Ch[11] <-> DI13/1600END input-bit maping/Digital input CH2-bit3
//     PlcTask Inputs/G_IO.arDI[13]/Ch[12] <-> DI13/1600END input-bit maping/Digital input CH2-bit4
//     PlcTask Inputs/G_IO.arDI[13]/Ch[13] <-> DI13/1600END input-bit maping/Digital input CH2-bit5
//     PlcTask Inputs/G_IO.arDI[13]/Ch[14] <-> DI13/1600END input-bit maping/Digital input CH2-bit6
//     PlcTask Inputs/G_IO.arDI[13]/Ch[15] <-> DI13/1600END input-bit maping/Digital input CH2-bit7
//     PlcTask Inputs/G_IO.arDI[13]/Ch[1] <-> DI13/1600END input-bit maping/Digital input CH1-bit1
//     PlcTask Inputs/G_IO.arDI[13]/Ch[2] <-> DI13/1600END input-bit maping/Digital input CH1-bit2
//     PlcTask Inputs/G_IO.arDI[13]/Ch[3] <-> DI13/1600END input-bit maping/Digital input CH1-bit3
//     PlcTask Inputs/G_IO.arDI[13]/Ch[4] <-> DI13/1600END input-bit maping/Digital input CH1-bit4
//     PlcTask Inputs/G_IO.arDI[13]/Ch[5] <-> DI13/1600END input-bit maping/Digital input CH1-bit5
//     PlcTask Inputs/G_IO.arDI[13]/Ch[6] <-> DI13/1600END input-bit maping/Digital input CH1-bit6
//     PlcTask Inputs/G_IO.arDI[13]/Ch[7] <-> DI13/1600END input-bit maping/Digital input CH1-bit7
//     PlcTask Inputs/G_IO.arDI[13]/Ch[8] <-> DI13/1600END input-bit maping/Digital input CH2-bit0
//     PlcTask Inputs/G_IO.arDI[13]/Ch[9] <-> DI13/1600END input-bit maping/Digital input CH2-bit1
//     PlcTask Inputs/G_IO.arDI[14]/Ch[0] <-> DI14/1600END input-bit maping/Digital input CH1-bit0
//     PlcTask Inputs/G_IO.arDI[14]/Ch[10] <-> DI14/1600END input-bit maping/Digital input CH2-bit2
//     PlcTask Inputs/G_IO.arDI[14]/Ch[11] <-> DI14/1600END input-bit maping/Digital input CH2-bit3
//     PlcTask Inputs/G_IO.arDI[14]/Ch[12] <-> DI14/1600END input-bit maping/Digital input CH2-bit4
//     PlcTask Inputs/G_IO.arDI[14]/Ch[13] <-> DI14/1600END input-bit maping/Digital input CH2-bit5
//     PlcTask Inputs/G_IO.arDI[14]/Ch[14] <-> DI14/1600END input-bit maping/Digital input CH2-bit6
//     PlcTask Inputs/G_IO.arDI[14]/Ch[15] <-> DI14/1600END input-bit maping/Digital input CH2-bit7
//     PlcTask Inputs/G_IO.arDI[14]/Ch[1] <-> DI14/1600END input-bit maping/Digital input CH1-bit1
//     PlcTask Inputs/G_IO.arDI[14]/Ch[2] <-> DI14/1600END input-bit maping/Digital input CH1-bit2
//     PlcTask Inputs/G_IO.arDI[14]/Ch[3] <-> DI14/1600END input-bit maping/Digital input CH1-bit3
//     PlcTask Inputs/G_IO.arDI[14]/Ch[4] <-> DI14/1600END input-bit maping/Digital input CH1-bit4
//     PlcTask Inputs/G_IO.arDI[14]/Ch[5] <-> DI14/1600END input-bit maping/Digital input CH1-bit5
//     PlcTask Inputs/G_IO.arDI[14]/Ch[6] <-> DI14/1600END input-bit maping/Digital input CH1-bit6
//     PlcTask Inputs/G_IO.arDI[14]/Ch[7] <-> DI14/1600END input-bit maping/Digital input CH1-bit7
//     PlcTask Inputs/G_IO.arDI[14]/Ch[8] <-> DI14/1600END input-bit maping/Digital input CH2-bit0
//     PlcTask Inputs/G_IO.arDI[14]/Ch[9] <-> DI14/1600END input-bit maping/Digital input CH2-bit1
//     PlcTask Inputs/G_IO.arDI[15]/Ch[0] <-> DI15/1600END input-bit maping/Digital input CH1-bit0
//     PlcTask Inputs/G_IO.arDI[15]/Ch[10] <-> DI15/1600END input-bit maping/Digital input CH2-bit2
//     PlcTask Inputs/G_IO.arDI[15]/Ch[11] <-> DI15/1600END input-bit maping/Digital input CH2-bit3
//     PlcTask Inputs/G_IO.arDI[15]/Ch[12] <-> DI15/1600END input-bit maping/Digital input CH2-bit4
//     PlcTask Inputs/G_IO.arDI[15]/Ch[13] <-> DI15/1600END input-bit maping/Digital input CH2-bit5
//     PlcTask Inputs/G_IO.arDI[15]/Ch[14] <-> DI15/1600END input-bit maping/Digital input CH2-bit6
//     PlcTask Inputs/G_IO.arDI[15]/Ch[15] <-> DI15/1600END input-bit maping/Digital input CH2-bit7
//     PlcTask Inputs/G_IO.arDI[15]/Ch[1] <-> DI15/1600END input-bit maping/Digital input CH1-bit1
//     PlcTask Inputs/G_IO.arDI[15]/Ch[2] <-> DI15/1600END input-bit maping/Digital input CH1-bit2
//     PlcTask Inputs/G_IO.arDI[15]/Ch[3] <-> DI15/1600END input-bit maping/Digital input CH1-bit3
//     PlcTask Inputs/G_IO.arDI[15]/Ch[4] <-> DI15/1600END input-bit maping/Digital input CH1-bit4
//     PlcTask Inputs/G_IO.arDI[15]/Ch[5] <-> DI15/1600END input-bit maping/Digital input CH1-bit5
//     PlcTask Inputs/G_IO.arDI[15]/Ch[6] <-> DI15/1600END input-bit maping/Digital input CH1-bit6
//     PlcTask Inputs/G_IO.arDI[15]/Ch[7] <-> DI15/1600END input-bit maping/Digital input CH1-bit7
//     PlcTask Inputs/G_IO.arDI[15]/Ch[8] <-> DI15/1600END input-bit maping/Digital input CH2-bit0
//     PlcTask Inputs/G_IO.arDI[15]/Ch[9] <-> DI15/1600END input-bit maping/Digital input CH2-bit1
//     PlcTask Outputs/G_IO.arDO[12]/Ch[0] <-> DO12/0016ETP Output-bit maping/Digital output CH1-bit0
//     PlcTask Outputs/G_IO.arDO[12]/Ch[10] <-> DO12/0016ETP Output-bit maping/Digital output CH2-bit2
//     PlcTask Outputs/G_IO.arDO[12]/Ch[11] <-> DO12/0016ETP Output-bit maping/Digital output CH2-bit3
//     PlcTask Outputs/G_IO.arDO[12]/Ch[12] <-> DO12/0016ETP Output-bit maping/Digital output CH2-bit4
//     PlcTask Outputs/G_IO.arDO[12]/Ch[13] <-> DO12/0016ETP Output-bit maping/Digital output CH2-bit5
//     PlcTask Outputs/G_IO.arDO[12]/Ch[14] <-> DO12/0016ETP Output-bit maping/Digital output CH2-bit6
//     PlcTask Outputs/G_IO.arDO[12]/Ch[15] <-> DO12/0016ETP Output-bit maping/Digital output CH2-bit7
//     PlcTask Outputs/G_IO.arDO[12]/Ch[1] <-> DO12/0016ETP Output-bit maping/Digital output CH1-bit1
//     PlcTask Outputs/G_IO.arDO[12]/Ch[2] <-> DO12/0016ETP Output-bit maping/Digital output CH1-bit2
//     PlcTask Outputs/G_IO.arDO[12]/Ch[3] <-> DO12/0016ETP Output-bit maping/Digital output CH1-bit3
//     PlcTask Outputs/G_IO.arDO[12]/Ch[4] <-> DO12/0016ETP Output-bit maping/Digital output CH1-bit4
//     PlcTask Outputs/G_IO.arDO[12]/Ch[5] <-> DO12/0016ETP Output-bit maping/Digital output CH1-bit5
//     PlcTask Outputs/G_IO.arDO[12]/Ch[6] <-> DO12/0016ETP Output-bit maping/Digital output CH1-bit6
//     PlcTask Outputs/G_IO.arDO[12]/Ch[7] <-> DO12/0016ETP Output-bit maping/Digital output CH1-bit7
//     PlcTask Outputs/G_IO.arDO[12]/Ch[8] <-> DO12/0016ETP Output-bit maping/Digital output CH2-bit0
//     PlcTask Outputs/G_IO.arDO[12]/Ch[9] <-> DO12/0016ETP Output-bit maping/Digital output CH2-bit1
//     PlcTask Outputs/G_IO.arDO[13]/Ch[0] <-> DO13/0016ETP Output-bit maping/Digital output CH1-bit0
//     PlcTask Outputs/G_IO.arDO[13]/Ch[10] <-> DO13/0016ETP Output-bit maping/Digital output CH2-bit2
//     PlcTask Outputs/G_IO.arDO[13]/Ch[11] <-> DO13/0016ETP Output-bit maping/Digital output CH2-bit3
//     PlcTask Outputs/G_IO.arDO[13]/Ch[12] <-> DO13/0016ETP Output-bit maping/Digital output CH2-bit4
//     PlcTask Outputs/G_IO.arDO[13]/Ch[13] <-> DO13/0016ETP Output-bit maping/Digital output CH2-bit5
//     PlcTask Outputs/G_IO.arDO[13]/Ch[14] <-> DO13/0016ETP Output-bit maping/Digital output CH2-bit6
//     PlcTask Outputs/G_IO.arDO[13]/Ch[15] <-> DO13/0016ETP Output-bit maping/Digital output CH2-bit7
//     PlcTask Outputs/G_IO.arDO[13]/Ch[1] <-> DO13/0016ETP Output-bit maping/Digital output CH1-bit1
//     PlcTask Outputs/G_IO.arDO[13]/Ch[2] <-> DO13/0016ETP Output-bit maping/Digital output CH1-bit2
//     PlcTask Outputs/G_IO.arDO[13]/Ch[3] <-> DO13/0016ETP Output-bit maping/Digital output CH1-bit3
//     PlcTask Outputs/G_IO.arDO[13]/Ch[4] <-> DO13/0016ETP Output-bit maping/Digital output CH1-bit4
//     PlcTask Outputs/G_IO.arDO[13]/Ch[5] <-> DO13/0016ETP Output-bit maping/Digital output CH1-bit5
//     PlcTask Outputs/G_IO.arDO[13]/Ch[6] <-> DO13/0016ETP Output-bit maping/Digital output CH1-bit6
//     PlcTask Outputs/G_IO.arDO[13]/Ch[7] <-> DO13/0016ETP Output-bit maping/Digital output CH1-bit7
//     PlcTask Outputs/G_IO.arDO[13]/Ch[8] <-> DO13/0016ETP Output-bit maping/Digital output CH2-bit0
//     PlcTask Outputs/G_IO.arDO[13]/Ch[9] <-> DO13/0016ETP Output-bit maping/Digital output CH2-bit1
//   kittingDeca/kittingDeca Instance <-> rem_wf/rem3_valve
//     PlcTask Outputs/G_IO.arDO[14]/Ch[0] <-> Module 1 (C2S-EC-24B)/Outputs/valve[1..4][0]
//     PlcTask Outputs/G_IO.arDO[14]/Ch[10] <-> Module 1 (C2S-EC-24B)/Outputs/valve[5..8][2]
//     PlcTask Outputs/G_IO.arDO[14]/Ch[11] <-> Module 1 (C2S-EC-24B)/Outputs/valve[5..8][3]
//     PlcTask Outputs/G_IO.arDO[14]/Ch[12] <-> Module 1 (C2S-EC-24B)/Outputs/valve[5..8][4]
//     PlcTask Outputs/G_IO.arDO[14]/Ch[13] <-> Module 1 (C2S-EC-24B)/Outputs/valve[5..8][5]
//     PlcTask Outputs/G_IO.arDO[14]/Ch[14] <-> Module 1 (C2S-EC-24B)/Outputs/valve[5..8][6]
//     PlcTask Outputs/G_IO.arDO[14]/Ch[15] <-> Module 1 (C2S-EC-24B)/Outputs/valve[5..8][7]
//     PlcTask Outputs/G_IO.arDO[14]/Ch[1] <-> Module 1 (C2S-EC-24B)/Outputs/valve[1..4][1]
//     PlcTask Outputs/G_IO.arDO[14]/Ch[2] <-> Module 1 (C2S-EC-24B)/Outputs/valve[1..4][2]
//     PlcTask Outputs/G_IO.arDO[14]/Ch[3] <-> Module 1 (C2S-EC-24B)/Outputs/valve[1..4][3]
//     PlcTask Outputs/G_IO.arDO[14]/Ch[4] <-> Module 1 (C2S-EC-24B)/Outputs/valve[1..4][4]
//     PlcTask Outputs/G_IO.arDO[14]/Ch[5] <-> Module 1 (C2S-EC-24B)/Outputs/valve[1..4][5]
//     PlcTask Outputs/G_IO.arDO[14]/Ch[6] <-> Module 1 (C2S-EC-24B)/Outputs/valve[1..4][6]
//     PlcTask Outputs/G_IO.arDO[14]/Ch[7] <-> Module 1 (C2S-EC-24B)/Outputs/valve[1..4][7]
//     PlcTask Outputs/G_IO.arDO[14]/Ch[8] <-> Module 1 (C2S-EC-24B)/Outputs/valve[5..8][0]
//     PlcTask Outputs/G_IO.arDO[14]/Ch[9] <-> Module 1 (C2S-EC-24B)/Outputs/valve[5..8][1]
//     PlcTask Outputs/G_IO.arDO[15]/Ch[0] <-> Module 1 (C2S-EC-24B)/Outputs/valve[9..12][0]
//     PlcTask Outputs/G_IO.arDO[15]/Ch[1] <-> Module 1 (C2S-EC-24B)/Outputs/valve[9..12][1]
//     PlcTask Outputs/G_IO.arDO[15]/Ch[2] <-> Module 1 (C2S-EC-24B)/Outputs/valve[9..12][2]
//     PlcTask Outputs/G_IO.arDO[15]/Ch[3] <-> Module 1 (C2S-EC-24B)/Outputs/valve[9..12][3]
//     PlcTask Outputs/G_IO.arDO[15]/Ch[4] <-> Module 1 (C2S-EC-24B)/Outputs/valve[9..12][4]
//     PlcTask Outputs/G_IO.arDO[15]/Ch[5] <-> Module 1 (C2S-EC-24B)/Outputs/valve[9..12][5]
//     PlcTask Outputs/G_IO.arDO[15]/Ch[6] <-> Module 1 (C2S-EC-24B)/Outputs/valve[9..12][6]
//     PlcTask Outputs/G_IO.arDO[15]/Ch[7] <-> Module 1 (C2S-EC-24B)/Outputs/valve[9..12][7]
//   kittingDeca/kittingDeca Instance <-> rem_wf/rem4_dio
//     PlcTask Inputs/G_IO.arDI[16]/Ch[0] <-> DI0/1600END input-bit maping/Digital input CH1-bit0
//     PlcTask Inputs/G_IO.arDI[16]/Ch[10] <-> DI0/1600END input-bit maping/Digital input CH2-bit2
//     PlcTask Inputs/G_IO.arDI[16]/Ch[11] <-> DI0/1600END input-bit maping/Digital input CH2-bit3
//     PlcTask Inputs/G_IO.arDI[16]/Ch[12] <-> DI0/1600END input-bit maping/Digital input CH2-bit4
//     PlcTask Inputs/G_IO.arDI[16]/Ch[13] <-> DI0/1600END input-bit maping/Digital input CH2-bit5
//     PlcTask Inputs/G_IO.arDI[16]/Ch[14] <-> DI0/1600END input-bit maping/Digital input CH2-bit6
//     PlcTask Inputs/G_IO.arDI[16]/Ch[15] <-> DI0/1600END input-bit maping/Digital input CH2-bit7
//     PlcTask Inputs/G_IO.arDI[16]/Ch[1] <-> DI0/1600END input-bit maping/Digital input CH1-bit1
//     PlcTask Inputs/G_IO.arDI[16]/Ch[2] <-> DI0/1600END input-bit maping/Digital input CH1-bit2
//     PlcTask Inputs/G_IO.arDI[16]/Ch[3] <-> DI0/1600END input-bit maping/Digital input CH1-bit3
//     PlcTask Inputs/G_IO.arDI[16]/Ch[4] <-> DI0/1600END input-bit maping/Digital input CH1-bit4
//     PlcTask Inputs/G_IO.arDI[16]/Ch[5] <-> DI0/1600END input-bit maping/Digital input CH1-bit5
//     PlcTask Inputs/G_IO.arDI[16]/Ch[6] <-> DI0/1600END input-bit maping/Digital input CH1-bit6
//     PlcTask Inputs/G_IO.arDI[16]/Ch[7] <-> DI0/1600END input-bit maping/Digital input CH1-bit7
//     PlcTask Inputs/G_IO.arDI[16]/Ch[8] <-> DI0/1600END input-bit maping/Digital input CH2-bit0
//     PlcTask Inputs/G_IO.arDI[16]/Ch[9] <-> DI0/1600END input-bit maping/Digital input CH2-bit1
//     PlcTask Inputs/G_IO.arDI[17]/Ch[0] <-> DI1/1600END input-bit maping/Digital input CH1-bit0
//     PlcTask Inputs/G_IO.arDI[17]/Ch[10] <-> DI1/1600END input-bit maping/Digital input CH2-bit2
//     PlcTask Inputs/G_IO.arDI[17]/Ch[11] <-> DI1/1600END input-bit maping/Digital input CH2-bit3
//     PlcTask Inputs/G_IO.arDI[17]/Ch[12] <-> DI1/1600END input-bit maping/Digital input CH2-bit4
//     PlcTask Inputs/G_IO.arDI[17]/Ch[13] <-> DI1/1600END input-bit maping/Digital input CH2-bit5
//     PlcTask Inputs/G_IO.arDI[17]/Ch[14] <-> DI1/1600END input-bit maping/Digital input CH2-bit6
//     PlcTask Inputs/G_IO.arDI[17]/Ch[15] <-> DI1/1600END input-bit maping/Digital input CH2-bit7
//     PlcTask Inputs/G_IO.arDI[17]/Ch[1] <-> DI1/1600END input-bit maping/Digital input CH1-bit1
//     PlcTask Inputs/G_IO.arDI[17]/Ch[2] <-> DI1/1600END input-bit maping/Digital input CH1-bit2
//     PlcTask Inputs/G_IO.arDI[17]/Ch[3] <-> DI1/1600END input-bit maping/Digital input CH1-bit3
//     PlcTask Inputs/G_IO.arDI[17]/Ch[4] <-> DI1/1600END input-bit maping/Digital input CH1-bit4
//     PlcTask Inputs/G_IO.arDI[17]/Ch[5] <-> DI1/1600END input-bit maping/Digital input CH1-bit5
//     PlcTask Inputs/G_IO.arDI[17]/Ch[6] <-> DI1/1600END input-bit maping/Digital input CH1-bit6
//     PlcTask Inputs/G_IO.arDI[17]/Ch[7] <-> DI1/1600END input-bit maping/Digital input CH1-bit7
//     PlcTask Inputs/G_IO.arDI[17]/Ch[8] <-> DI1/1600END input-bit maping/Digital input CH2-bit0
//     PlcTask Inputs/G_IO.arDI[17]/Ch[9] <-> DI1/1600END input-bit maping/Digital input CH2-bit1
//     PlcTask Inputs/G_IO.arDI[18]/Ch[0] <-> DI2/1600END input-bit maping/Digital input CH1-bit0
//     PlcTask Inputs/G_IO.arDI[18]/Ch[10] <-> DI2/1600END input-bit maping/Digital input CH2-bit2
//     PlcTask Inputs/G_IO.arDI[18]/Ch[11] <-> DI2/1600END input-bit maping/Digital input CH2-bit3
//     PlcTask Inputs/G_IO.arDI[18]/Ch[12] <-> DI2/1600END input-bit maping/Digital input CH2-bit4
//     PlcTask Inputs/G_IO.arDI[18]/Ch[13] <-> DI2/1600END input-bit maping/Digital input CH2-bit5
//     PlcTask Inputs/G_IO.arDI[18]/Ch[14] <-> DI2/1600END input-bit maping/Digital input CH2-bit6
//     PlcTask Inputs/G_IO.arDI[18]/Ch[15] <-> DI2/1600END input-bit maping/Digital input CH2-bit7
//     PlcTask Inputs/G_IO.arDI[18]/Ch[1] <-> DI2/1600END input-bit maping/Digital input CH1-bit1
//     PlcTask Inputs/G_IO.arDI[18]/Ch[2] <-> DI2/1600END input-bit maping/Digital input CH1-bit2
//     PlcTask Inputs/G_IO.arDI[18]/Ch[3] <-> DI2/1600END input-bit maping/Digital input CH1-bit3
//     PlcTask Inputs/G_IO.arDI[18]/Ch[4] <-> DI2/1600END input-bit maping/Digital input CH1-bit4
//     PlcTask Inputs/G_IO.arDI[18]/Ch[5] <-> DI2/1600END input-bit maping/Digital input CH1-bit5
//     PlcTask Inputs/G_IO.arDI[18]/Ch[6] <-> DI2/1600END input-bit maping/Digital input CH1-bit6
//     PlcTask Inputs/G_IO.arDI[18]/Ch[7] <-> DI2/1600END input-bit maping/Digital input CH1-bit7
//     PlcTask Inputs/G_IO.arDI[18]/Ch[8] <-> DI2/1600END input-bit maping/Digital input CH2-bit0
//     PlcTask Inputs/G_IO.arDI[18]/Ch[9] <-> DI2/1600END input-bit maping/Digital input CH2-bit1
//     PlcTask Inputs/G_IO.arDI[19]/Ch[0] <-> DI3/1600END input-bit maping/Digital input CH1-bit0
//     PlcTask Inputs/G_IO.arDI[19]/Ch[10] <-> DI3/1600END input-bit maping/Digital input CH2-bit2
//     PlcTask Inputs/G_IO.arDI[19]/Ch[11] <-> DI3/1600END input-bit maping/Digital input CH2-bit3
//     PlcTask Inputs/G_IO.arDI[19]/Ch[12] <-> DI3/1600END input-bit maping/Digital input CH2-bit4
//     PlcTask Inputs/G_IO.arDI[19]/Ch[13] <-> DI3/1600END input-bit maping/Digital input CH2-bit5
//     PlcTask Inputs/G_IO.arDI[19]/Ch[14] <-> DI3/1600END input-bit maping/Digital input CH2-bit6
//     PlcTask Inputs/G_IO.arDI[19]/Ch[15] <-> DI3/1600END input-bit maping/Digital input CH2-bit7
//     PlcTask Inputs/G_IO.arDI[19]/Ch[1] <-> DI3/1600END input-bit maping/Digital input CH1-bit1
//     PlcTask Inputs/G_IO.arDI[19]/Ch[2] <-> DI3/1600END input-bit maping/Digital input CH1-bit2
//     PlcTask Inputs/G_IO.arDI[19]/Ch[3] <-> DI3/1600END input-bit maping/Digital input CH1-bit3
//     PlcTask Inputs/G_IO.arDI[19]/Ch[4] <-> DI3/1600END input-bit maping/Digital input CH1-bit4
//     PlcTask Inputs/G_IO.arDI[19]/Ch[5] <-> DI3/1600END input-bit maping/Digital input CH1-bit5
//     PlcTask Inputs/G_IO.arDI[19]/Ch[6] <-> DI3/1600END input-bit maping/Digital input CH1-bit6
//     PlcTask Inputs/G_IO.arDI[19]/Ch[7] <-> DI3/1600END input-bit maping/Digital input CH1-bit7
//     PlcTask Inputs/G_IO.arDI[19]/Ch[8] <-> DI3/1600END input-bit maping/Digital input CH2-bit0
//     PlcTask Inputs/G_IO.arDI[19]/Ch[9] <-> DI3/1600END input-bit maping/Digital input CH2-bit1
//     PlcTask Outputs/G_IO.arDO[16]/Ch[0] <-> DO0/0016ETP Output-bit maping/Digital output CH1-bit0
//     PlcTask Outputs/G_IO.arDO[16]/Ch[10] <-> DO0/0016ETP Output-bit maping/Digital output CH2-bit2
//     PlcTask Outputs/G_IO.arDO[16]/Ch[11] <-> DO0/0016ETP Output-bit maping/Digital output CH2-bit3
//     PlcTask Outputs/G_IO.arDO[16]/Ch[12] <-> DO0/0016ETP Output-bit maping/Digital output CH2-bit4
//     PlcTask Outputs/G_IO.arDO[16]/Ch[13] <-> DO0/0016ETP Output-bit maping/Digital output CH2-bit5
//     PlcTask Outputs/G_IO.arDO[16]/Ch[14] <-> DO0/0016ETP Output-bit maping/Digital output CH2-bit6
//     PlcTask Outputs/G_IO.arDO[16]/Ch[15] <-> DO0/0016ETP Output-bit maping/Digital output CH2-bit7
//     PlcTask Outputs/G_IO.arDO[16]/Ch[1] <-> DO0/0016ETP Output-bit maping/Digital output CH1-bit1
//     PlcTask Outputs/G_IO.arDO[16]/Ch[2] <-> DO0/0016ETP Output-bit maping/Digital output CH1-bit2
//     PlcTask Outputs/G_IO.arDO[16]/Ch[3] <-> DO0/0016ETP Output-bit maping/Digital output CH1-bit3
//     PlcTask Outputs/G_IO.arDO[16]/Ch[4] <-> DO0/0016ETP Output-bit maping/Digital output CH1-bit4
//     PlcTask Outputs/G_IO.arDO[16]/Ch[5] <-> DO0/0016ETP Output-bit maping/Digital output CH1-bit5
//     PlcTask Outputs/G_IO.arDO[16]/Ch[6] <-> DO0/0016ETP Output-bit maping/Digital output CH1-bit6
//     PlcTask Outputs/G_IO.arDO[16]/Ch[7] <-> DO0/0016ETP Output-bit maping/Digital output CH1-bit7
//     PlcTask Outputs/G_IO.arDO[16]/Ch[8] <-> DO0/0016ETP Output-bit maping/Digital output CH2-bit0
//     PlcTask Outputs/G_IO.arDO[16]/Ch[9] <-> DO0/0016ETP Output-bit maping/Digital output CH2-bit1
//     PlcTask Outputs/G_IO.arDO[17]/Ch[0] <-> DO1/0016ETP Output-bit maping/Digital output CH1-bit0
//     PlcTask Outputs/G_IO.arDO[17]/Ch[10] <-> DO1/0016ETP Output-bit maping/Digital output CH2-bit2
//     PlcTask Outputs/G_IO.arDO[17]/Ch[11] <-> DO1/0016ETP Output-bit maping/Digital output CH2-bit3
//     PlcTask Outputs/G_IO.arDO[17]/Ch[12] <-> DO1/0016ETP Output-bit maping/Digital output CH2-bit4
//     PlcTask Outputs/G_IO.arDO[17]/Ch[13] <-> DO1/0016ETP Output-bit maping/Digital output CH2-bit5
//     PlcTask Outputs/G_IO.arDO[17]/Ch[14] <-> DO1/0016ETP Output-bit maping/Digital output CH2-bit6
//     PlcTask Outputs/G_IO.arDO[17]/Ch[15] <-> DO1/0016ETP Output-bit maping/Digital output CH2-bit7
//     PlcTask Outputs/G_IO.arDO[17]/Ch[1] <-> DO1/0016ETP Output-bit maping/Digital output CH1-bit1
//     PlcTask Outputs/G_IO.arDO[17]/Ch[2] <-> DO1/0016ETP Output-bit maping/Digital output CH1-bit2
//     PlcTask Outputs/G_IO.arDO[17]/Ch[3] <-> DO1/0016ETP Output-bit maping/Digital output CH1-bit3
//     PlcTask Outputs/G_IO.arDO[17]/Ch[4] <-> DO1/0016ETP Output-bit maping/Digital output CH1-bit4
//     PlcTask Outputs/G_IO.arDO[17]/Ch[5] <-> DO1/0016ETP Output-bit maping/Digital output CH1-bit5
//     PlcTask Outputs/G_IO.arDO[17]/Ch[6] <-> DO1/0016ETP Output-bit maping/Digital output CH1-bit6
//     PlcTask Outputs/G_IO.arDO[17]/Ch[7] <-> DO1/0016ETP Output-bit maping/Digital output CH1-bit7
//     PlcTask Outputs/G_IO.arDO[17]/Ch[8] <-> DO1/0016ETP Output-bit maping/Digital output CH2-bit0
//     PlcTask Outputs/G_IO.arDO[17]/Ch[9] <-> DO1/0016ETP Output-bit maping/Digital output CH2-bit1
//   kittingDeca/kittingDeca Instance <-> rem_wf/rem4_valve
//     PlcTask Outputs/G_IO.arDO[18]/Ch[0] <-> Module 1 (C2S-EC-24B)/Outputs/valve[1..4][0]
//     PlcTask Outputs/G_IO.arDO[18]/Ch[10] <-> Module 1 (C2S-EC-24B)/Outputs/valve[5..8][2]
//     PlcTask Outputs/G_IO.arDO[18]/Ch[11] <-> Module 1 (C2S-EC-24B)/Outputs/valve[5..8][3]
//     PlcTask Outputs/G_IO.arDO[18]/Ch[12] <-> Module 1 (C2S-EC-24B)/Outputs/valve[5..8][4]
//     PlcTask Outputs/G_IO.arDO[18]/Ch[13] <-> Module 1 (C2S-EC-24B)/Outputs/valve[5..8][5]
//     PlcTask Outputs/G_IO.arDO[18]/Ch[14] <-> Module 1 (C2S-EC-24B)/Outputs/valve[5..8][6]
//     PlcTask Outputs/G_IO.arDO[18]/Ch[15] <-> Module 1 (C2S-EC-24B)/Outputs/valve[5..8][7]
//     PlcTask Outputs/G_IO.arDO[18]/Ch[1] <-> Module 1 (C2S-EC-24B)/Outputs/valve[1..4][1]
//     PlcTask Outputs/G_IO.arDO[18]/Ch[2] <-> Module 1 (C2S-EC-24B)/Outputs/valve[1..4][2]
//     PlcTask Outputs/G_IO.arDO[18]/Ch[3] <-> Module 1 (C2S-EC-24B)/Outputs/valve[1..4][3]
//     PlcTask Outputs/G_IO.arDO[18]/Ch[4] <-> Module 1 (C2S-EC-24B)/Outputs/valve[1..4][4]
//     PlcTask Outputs/G_IO.arDO[18]/Ch[5] <-> Module 1 (C2S-EC-24B)/Outputs/valve[1..4][5]
//     PlcTask Outputs/G_IO.arDO[18]/Ch[6] <-> Module 1 (C2S-EC-24B)/Outputs/valve[1..4][6]
//     PlcTask Outputs/G_IO.arDO[18]/Ch[7] <-> Module 1 (C2S-EC-24B)/Outputs/valve[1..4][7]
//     PlcTask Outputs/G_IO.arDO[18]/Ch[8] <-> Module 1 (C2S-EC-24B)/Outputs/valve[5..8][0]
//     PlcTask Outputs/G_IO.arDO[18]/Ch[9] <-> Module 1 (C2S-EC-24B)/Outputs/valve[5..8][1]
//     PlcTask Outputs/G_IO.arDO[19]/Ch[0] <-> Module 1 (C2S-EC-24B)/Outputs/valve[9..12][0]
//     PlcTask Outputs/G_IO.arDO[19]/Ch[1] <-> Module 1 (C2S-EC-24B)/Outputs/valve[9..12][1]
//     PlcTask Outputs/G_IO.arDO[19]/Ch[2] <-> Module 1 (C2S-EC-24B)/Outputs/valve[9..12][2]
//     PlcTask Outputs/G_IO.arDO[19]/Ch[3] <-> Module 1 (C2S-EC-24B)/Outputs/valve[9..12][3]
//     PlcTask Outputs/G_IO.arDO[19]/Ch[4] <-> Module 1 (C2S-EC-24B)/Outputs/valve[9..12][4]
//     PlcTask Outputs/G_IO.arDO[19]/Ch[5] <-> Module 1 (C2S-EC-24B)/Outputs/valve[9..12][5]
//     PlcTask Outputs/G_IO.arDO[19]/Ch[6] <-> Module 1 (C2S-EC-24B)/Outputs/valve[9..12][6]
//     PlcTask Outputs/G_IO.arDO[19]/Ch[7] <-> Module 1 (C2S-EC-24B)/Outputs/valve[9..12][7]
//   kittingDeca/kittingDeca Instance <-> rem_wf/rem5_dio
//     PlcTask Inputs/G_IO.arDI[20]/Ch[0] <-> DI0/1600END input-bit maping/Digital input CH1-bit0
//     PlcTask Inputs/G_IO.arDI[20]/Ch[10] <-> DI0/1600END input-bit maping/Digital input CH2-bit2
//     PlcTask Inputs/G_IO.arDI[20]/Ch[11] <-> DI0/1600END input-bit maping/Digital input CH2-bit3
//     PlcTask Inputs/G_IO.arDI[20]/Ch[12] <-> DI0/1600END input-bit maping/Digital input CH2-bit4
//     PlcTask Inputs/G_IO.arDI[20]/Ch[13] <-> DI0/1600END input-bit maping/Digital input CH2-bit5
//     PlcTask Inputs/G_IO.arDI[20]/Ch[14] <-> DI0/1600END input-bit maping/Digital input CH2-bit6
//     PlcTask Inputs/G_IO.arDI[20]/Ch[15] <-> DI0/1600END input-bit maping/Digital input CH2-bit7
//     PlcTask Inputs/G_IO.arDI[20]/Ch[1] <-> DI0/1600END input-bit maping/Digital input CH1-bit1
//     PlcTask Inputs/G_IO.arDI[20]/Ch[2] <-> DI0/1600END input-bit maping/Digital input CH1-bit2
//     PlcTask Inputs/G_IO.arDI[20]/Ch[3] <-> DI0/1600END input-bit maping/Digital input CH1-bit3
//     PlcTask Inputs/G_IO.arDI[20]/Ch[4] <-> DI0/1600END input-bit maping/Digital input CH1-bit4
//     PlcTask Inputs/G_IO.arDI[20]/Ch[5] <-> DI0/1600END input-bit maping/Digital input CH1-bit5
//     PlcTask Inputs/G_IO.arDI[20]/Ch[6] <-> DI0/1600END input-bit maping/Digital input CH1-bit6
//     PlcTask Inputs/G_IO.arDI[20]/Ch[7] <-> DI0/1600END input-bit maping/Digital input CH1-bit7
//     PlcTask Inputs/G_IO.arDI[20]/Ch[8] <-> DI0/1600END input-bit maping/Digital input CH2-bit0
//     PlcTask Inputs/G_IO.arDI[20]/Ch[9] <-> DI0/1600END input-bit maping/Digital input CH2-bit1
//     PlcTask Inputs/G_IO.arDI[21]/Ch[0] <-> DI1/1600END input-bit maping/Digital input CH1-bit0
//     PlcTask Inputs/G_IO.arDI[21]/Ch[10] <-> DI1/1600END input-bit maping/Digital input CH2-bit2
//     PlcTask Inputs/G_IO.arDI[21]/Ch[11] <-> DI1/1600END input-bit maping/Digital input CH2-bit3
//     PlcTask Inputs/G_IO.arDI[21]/Ch[12] <-> DI1/1600END input-bit maping/Digital input CH2-bit4
//     PlcTask Inputs/G_IO.arDI[21]/Ch[13] <-> DI1/1600END input-bit maping/Digital input CH2-bit5
//     PlcTask Inputs/G_IO.arDI[21]/Ch[14] <-> DI1/1600END input-bit maping/Digital input CH2-bit6
//     PlcTask Inputs/G_IO.arDI[21]/Ch[15] <-> DI1/1600END input-bit maping/Digital input CH2-bit7
//     PlcTask Inputs/G_IO.arDI[21]/Ch[1] <-> DI1/1600END input-bit maping/Digital input CH1-bit1
//     PlcTask Inputs/G_IO.arDI[21]/Ch[2] <-> DI1/1600END input-bit maping/Digital input CH1-bit2
//     PlcTask Inputs/G_IO.arDI[21]/Ch[3] <-> DI1/1600END input-bit maping/Digital input CH1-bit3
//     PlcTask Inputs/G_IO.arDI[21]/Ch[4] <-> DI1/1600END input-bit maping/Digital input CH1-bit4
//     PlcTask Inputs/G_IO.arDI[21]/Ch[5] <-> DI1/1600END input-bit maping/Digital input CH1-bit5
//     PlcTask Inputs/G_IO.arDI[21]/Ch[6] <-> DI1/1600END input-bit maping/Digital input CH1-bit6
//     PlcTask Inputs/G_IO.arDI[21]/Ch[7] <-> DI1/1600END input-bit maping/Digital input CH1-bit7
//     PlcTask Inputs/G_IO.arDI[21]/Ch[8] <-> DI1/1600END input-bit maping/Digital input CH2-bit0
//     PlcTask Inputs/G_IO.arDI[21]/Ch[9] <-> DI1/1600END input-bit maping/Digital input CH2-bit1
//     PlcTask Inputs/G_IO.arDI[22]/Ch[0] <-> DI2/1600END input-bit maping/Digital input CH1-bit0
//     PlcTask Inputs/G_IO.arDI[22]/Ch[10] <-> DI2/1600END input-bit maping/Digital input CH2-bit2
//     PlcTask Inputs/G_IO.arDI[22]/Ch[11] <-> DI2/1600END input-bit maping/Digital input CH2-bit3
//     PlcTask Inputs/G_IO.arDI[22]/Ch[12] <-> DI2/1600END input-bit maping/Digital input CH2-bit4
//     PlcTask Inputs/G_IO.arDI[22]/Ch[13] <-> DI2/1600END input-bit maping/Digital input CH2-bit5
//     PlcTask Inputs/G_IO.arDI[22]/Ch[14] <-> DI2/1600END input-bit maping/Digital input CH2-bit6
//     PlcTask Inputs/G_IO.arDI[22]/Ch[15] <-> DI2/1600END input-bit maping/Digital input CH2-bit7
//     PlcTask Inputs/G_IO.arDI[22]/Ch[1] <-> DI2/1600END input-bit maping/Digital input CH1-bit1
//     PlcTask Inputs/G_IO.arDI[22]/Ch[2] <-> DI2/1600END input-bit maping/Digital input CH1-bit2
//     PlcTask Inputs/G_IO.arDI[22]/Ch[3] <-> DI2/1600END input-bit maping/Digital input CH1-bit3
//     PlcTask Inputs/G_IO.arDI[22]/Ch[4] <-> DI2/1600END input-bit maping/Digital input CH1-bit4
//     PlcTask Inputs/G_IO.arDI[22]/Ch[5] <-> DI2/1600END input-bit maping/Digital input CH1-bit5
//     PlcTask Inputs/G_IO.arDI[22]/Ch[6] <-> DI2/1600END input-bit maping/Digital input CH1-bit6
//     PlcTask Inputs/G_IO.arDI[22]/Ch[7] <-> DI2/1600END input-bit maping/Digital input CH1-bit7
//     PlcTask Inputs/G_IO.arDI[22]/Ch[8] <-> DI2/1600END input-bit maping/Digital input CH2-bit0
//     PlcTask Inputs/G_IO.arDI[22]/Ch[9] <-> DI2/1600END input-bit maping/Digital input CH2-bit1
//     PlcTask Inputs/G_IO.arDI[23]/Ch[0] <-> DI3/1600END input-bit maping/Digital input CH1-bit0
//     PlcTask Inputs/G_IO.arDI[23]/Ch[10] <-> DI3/1600END input-bit maping/Digital input CH2-bit2
//     PlcTask Inputs/G_IO.arDI[23]/Ch[11] <-> DI3/1600END input-bit maping/Digital input CH2-bit3
//     PlcTask Inputs/G_IO.arDI[23]/Ch[12] <-> DI3/1600END input-bit maping/Digital input CH2-bit4
//     PlcTask Inputs/G_IO.arDI[23]/Ch[13] <-> DI3/1600END input-bit maping/Digital input CH2-bit5
//     PlcTask Inputs/G_IO.arDI[23]/Ch[14] <-> DI3/1600END input-bit maping/Digital input CH2-bit6
//     PlcTask Inputs/G_IO.arDI[23]/Ch[15] <-> DI3/1600END input-bit maping/Digital input CH2-bit7
//     PlcTask Inputs/G_IO.arDI[23]/Ch[1] <-> DI3/1600END input-bit maping/Digital input CH1-bit1
//     PlcTask Inputs/G_IO.arDI[23]/Ch[2] <-> DI3/1600END input-bit maping/Digital input CH1-bit2
//     PlcTask Inputs/G_IO.arDI[23]/Ch[3] <-> DI3/1600END input-bit maping/Digital input CH1-bit3
//     PlcTask Inputs/G_IO.arDI[23]/Ch[4] <-> DI3/1600END input-bit maping/Digital input CH1-bit4
//     PlcTask Inputs/G_IO.arDI[23]/Ch[5] <-> DI3/1600END input-bit maping/Digital input CH1-bit5
//     PlcTask Inputs/G_IO.arDI[23]/Ch[6] <-> DI3/1600END input-bit maping/Digital input CH1-bit6
//     PlcTask Inputs/G_IO.arDI[23]/Ch[7] <-> DI3/1600END input-bit maping/Digital input CH1-bit7
//     PlcTask Inputs/G_IO.arDI[23]/Ch[8] <-> DI3/1600END input-bit maping/Digital input CH2-bit0
//     PlcTask Inputs/G_IO.arDI[23]/Ch[9] <-> DI3/1600END input-bit maping/Digital input CH2-bit1
//     PlcTask Outputs/G_IO.arDO[20]/Ch[0] <-> DO0/0016ETP Output-bit maping/Digital output CH1-bit0
//     PlcTask Outputs/G_IO.arDO[20]/Ch[10] <-> DO0/0016ETP Output-bit maping/Digital output CH2-bit2
